gfCNCPoint1[16841] = {X 353.0465, Y 35.4906, Z -1.3333, A 0.000, B 0.000, C 0.000 }
gfCNCPoint1[16842] = {X 354.2270, Y 34.3409, Z -1.3333, A 0.000, B 0.000, C 0.000 }
gfCNCPoint1[16843] = {X 355.2487, Y 33.0481, Z -1.3333, A 0.000, B 0.000, C 0.000 }
gfCNCPoint1[16844] = {X 356.0944, Y 31.6339, Z -1.3333, A 0.000, B 0.000, C 0.000 }
gfCNCPoint1[16845] = {X 356.7500, Y 30.1221, Z -1.3333, A 0.000, B 0.000, C 0.000 }
gfCNCPoint1[16846] = {X 357.2044, Y 28.5381, Z -1.3333, A 0.000, B 0.000, C 0.000 }
gfCNCPoint1[16847] = {X 357.4826, Y 26.8196, Z -1.3333, A 0.000, B 0.000, C 0.000 }
gfCNCPoint1[16848] = {X 357.5960, Y 25.0823, Z -1.3333, A 0.000, B 0.000, C 0.000 }
gfCNCPoint1[16849] = {X 357.5434, Y 23.3422, Z -1.3333, A 0.000, B 0.000, C 0.000 }
gfCNCPoint1[16850] = {X 357.3254, Y 21.6150, Z -1.3333, A 0.000, B 0.000, C 0.000 }
gfCNCPoint1[16851] = {X 356.9800, Y 20.1274, Z -1.3333, A 0.000, B 0.000, C 0.000 }
gfCNCPoint1[16852] = {X 356.4533, Y 18.6940, Z -1.3333, A 0.000, B 0.000, C 0.000 }
gfCNCPoint1[16853] = {X 355.7534, Y 17.3367, Z -1.3333, A 0.000, B 0.000, C 0.000 }
gfCNCPoint1[16854] = {X 354.8909, Y 16.0764, Z -1.3333, A 0.000, B 0.000, C 0.000 }
gfCNCPoint1[16855] = {X 353.9742, Y 15.0542, Z -1.3333, A 0.000, B 0.000, C 0.000 }
gfCNCPoint1[16856] = {X 352.9205, Y 14.1738, Z -1.3333, A 0.000, B 0.000, C 0.000 }
gfCNCPoint1[16857] = {X 351.7516, Y 13.4534, Z -1.3333, A 0.000, B 0.000, C 0.000 }
gfCNCPoint1[16858] = {X 350.4916, Y 12.9079, Z -1.3333, A 0.000, B 0.000, C 0.000 }
gfCNCPoint1[16859] = {X 349.1664, Y 12.5485, Z -1.3333, A 0.000, B 0.000, C 0.000 }
gfCNCPoint1[16860] = {X 347.3712, Y 12.3248, Z -1.3333, A 0.000, B 0.000, C 0.000 }
gfCNCPoint1[16861] = {X 345.5623, Y 12.3395, Z -1.3333, A 0.000, B 0.000, C 0.000 }
gfCNCPoint1[16862] = {X 343.7710, Y 12.5924, Z -1.3333, A 0.000, B 0.000, C 0.000 }
gfCNCPoint1[16863] = {X 342.0287, Y 13.0789, Z -1.3333, A 0.000, B 0.000, C 0.000 }
gfCNCPoint1[16864] = {X 340.3656, Y 13.7908, Z -1.3333, A 0.000, B 0.000, C 0.000 }
gfCNCPoint1[16865] = {X 338.8108, Y 14.7154, Z -1.3333, A 0.000, B 0.000, C 0.000 }
gfCNCPoint1[16866] = {X 338.7172, Y 14.7804, Z -1.3333, A 0.000, B 0.000, C 0.000 }
gfCNCPoint1[16867] = {X 338.6242, Y 14.8461, Z -1.3333, A 0.000, B 0.000, C 0.000 }
gfCNCPoint1[16868] = {X 338.6379, Y 15.0619, Z -1.3333, A 0.000, B 0.000, C 0.000 }
gfCNCPoint1[16869] = {X 338.5598, Y 16.0346, Z -1.3333, A 0.000, B 0.000, C 0.000 }
gfCNCPoint1[16870] = {X 338.2486, Y 16.9596, Z -1.3333, A 0.000, B 0.000, C 0.000 }
gfCNCPoint1[16871] = {X 337.7226, Y 17.7816, Z -1.3333, A 0.000, B 0.000, C 0.000 }
gfCNCPoint1[16872] = {X 337.0132, Y 18.4518, Z -1.3333, A 0.000, B 0.000, C 0.000 }
gfCNCPoint1[16873] = {X 336.3278, Y 18.9560, Z -1.3333, A 0.000, B 0.000, C 0.000 }
gfCNCPoint1[16874] = {X 335.5713, Y 19.3817, Z -1.3333, A 0.000, B 0.000, C 0.000 }
gfCNCPoint1[16875] = {X 334.7407, Y 19.6341, Z -1.3333, A 0.000, B 0.000, C 0.000 }
gfCNCPoint1[16876] = {X 333.8753, Y 19.7014, Z -1.3333, A 0.000, B 0.000, C 0.000 }
gfCNCPoint1[16877] = {X 333.0157, Y 19.5804, Z -1.3333, A 0.000, B 0.000, C 0.000 }
gfCNCPoint1[16878] = {X 332.2025, Y 19.2768, Z -1.3333, A 0.000, B 0.000, C 0.000 }
gfCNCPoint1[16879] = {X 331.4739, Y 18.8049, Z -1.3333, A 0.000, B 0.000, C 0.000 }
gfCNCPoint1[16880] = {X 330.8643, Y 18.1870, Z -1.3333, A 0.000, B 0.000, C 0.000 }
gfCNCPoint1[16881] = {X 330.4023, Y 17.4521, Z -1.3333, A 0.000, B 0.000, C 0.000 }
gfCNCPoint1[16882] = {X 326.8820, Y 10.2103, Z -1.3333, A 0.000, B 0.000, C 0.000 }
gfCNCPoint1[16883] = {X 326.5719, Y 9.3163, Z -1.3333, A 0.000, B 0.000, C 0.000 }
gfCNCPoint1[16884] = {X 326.4804, Y 8.3746, Z -1.3333, A 0.000, B 0.000, C 0.000 }
gfCNCPoint1[16885] = {X 326.6127, Y 7.4376, Z -1.3333, A 0.000, B 0.000, C 0.000 }
gfCNCPoint1[16886] = {X 326.9614, Y 6.5580, Z -1.3333, A 0.000, B 0.000, C 0.000 }
gfCNCPoint1[16887] = {X 327.5070, Y 5.7849, Z -1.3333, A 0.000, B 0.000, C 0.000 }
gfCNCPoint1[16888] = {X 328.2189, Y 5.1616, Z -1.3333, A 0.000, B 0.000, C 0.000 }
gfCNCPoint1[16889] = {X 328.8880, Y 4.7034, Z -1.3333, A 0.000, B 0.000, C 0.000 }
gfCNCPoint1[16890] = {X 329.7043, Y 4.2813, Z -1.3333, A 0.000, B 0.000, C 0.000 }
gfCNCPoint1[16891] = {X 330.5954, Y 4.0567, Z -1.3333, A 0.000, B 0.000, C 0.000 }
gfCNCPoint1[16892] = {X 331.5142, Y 4.0413, Z -1.3333, A 0.000, B 0.000, C 0.000 }
gfCNCPoint1[16893] = {X 332.4122, Y 4.2361, Z -1.3333, A 0.000, B 0.000, C 0.000 }
gfCNCPoint1[16894] = {X 332.5467, Y 4.2834, Z -1.3333, A 0.000, B 0.000, C 0.000 }
gfCNCPoint1[16895] = {X 332.6264, Y 4.2354, Z -1.3333, A 0.000, B 0.000, C 0.000 }
gfCNCPoint1[16896] = {X 332.7062, Y 4.1876, Z -1.3333, A 0.000, B 0.000, C 0.000 }
gfCNCPoint1[16897] = {X 334.1618, Y 3.3772, Z -1.3333, A 0.000, B 0.000, C 0.000 }
gfCNCPoint1[16898] = {X 335.6629, Y 2.6547, Z -1.3333, A 0.000, B 0.000, C 0.000 }
gfCNCPoint1[16899] = {X 336.0092, Y 2.5006, Z -1.3333, A 0.000, B 0.000, C 0.000 }
gfCNCPoint1[16900] = {X 338.0805, Y 1.6925, Z -1.3333, A 0.000, B 0.000, C 0.000 }
gfCNCPoint1[16901] = {X 340.2133, Y 1.0646, Z -1.3333, A 0.000, B 0.000, C 0.000 }
gfCNCPoint1[16902] = {X 342.3920, Y 0.6215, Z -1.3333, A 0.000, B 0.000, C 0.000 }
gfCNCPoint1[16903] = {X 344.6007, Y 0.3665, Z -1.3333, A 0.000, B 0.000, C 0.000 }
gfCNCPoint1[16904] = {X 346.8231, Y 0.3014, Z -1.3333, A 0.000, B 0.000, C 0.000 }
gfCNCPoint1[16905] = {X 349.0429, Y 0.4266, Z -1.3333, A 0.000, B 0.000, C 0.000 }
gfCNCPoint1[16906] = {X 351.2438, Y 0.7414, Z -1.3333, A 0.000, B 0.000, C 0.000 }
gfCNCPoint1[16907] = {X 351.5273, Y 0.7937, Z -1.3333, A 0.000, B 0.000, C 0.000 }
gfCNCPoint1[16908] = {X 352.2677, Y -3.2186, Z -1.3333, A 0.000, B 0.000, C 0.000 }
gfCNCPoint1[16909] = {X 352.2677, Y -3.2186, Z 1.6667, A 0.000, B 0.000, C 0.000 }
gfCNCPoint1[16910] = {X 352.2677, Y -3.2186, Z 11.0000, A 0.000, B 0.000, C 0.000 }
gfCNCPoint1[16911] = {X 606.0428, Y 42.9012, Z 11.0000, A 0.000, B 0.000, C 0.000 }
gfCNCPoint1[16912] = {X 606.0428, Y 42.9012, Z 1.6667, A 0.000, B 0.000, C 0.000 }
gfCNCPoint1[16913] = {X 606.0428, Y 42.9012, Z -1.3333, A 0.000, B 0.000, C 0.000 }
gfCNCPoint1[16914] = {X 603.6965, Y 47.0770, Z -1.3333, A 0.000, B 0.000, C 0.000 }
gfCNCPoint1[16915] = {X 603.6310, Y 47.1895, Z -1.3333, A 0.000, B 0.000, C 0.000 }
gfCNCPoint1[16916] = {X 603.5620, Y 47.2999, Z -1.3333, A 0.000, B 0.000, C 0.000 }
gfCNCPoint1[16917] = {X 603.0356, Y 47.9602, Z -1.3333, A 0.000, B 0.000, C 0.000 }
gfCNCPoint1[16918] = {X 602.3888, Y 48.5030, Z -1.3333, A 0.000, B 0.000, C 0.000 }
gfCNCPoint1[16919] = {X 601.6472, Y 48.9070, Z -1.3333, A 0.000, B 0.000, C 0.000 }
gfCNCPoint1[16920] = {X 600.8403, Y 49.1559, Z -1.3333, A 0.000, B 0.000, C 0.000 }
gfCNCPoint1[16921] = {X 600.0000, Y 49.2400, Z -1.3333, A 0.000, B 0.000, C 0.000 }
gfCNCPoint1[16922] = {X 593.5565, Y 49.2400, Z -1.3333, A 0.000, B 0.000, C 0.000 }
gfCNCPoint1[16923] = {X 592.6130, Y 49.1337, Z -1.3333, A 0.000, B 0.000, C 0.000 }
gfCNCPoint1[16924] = {X 591.7169, Y 48.8201, Z -1.3333, A 0.000, B 0.000, C 0.000 }
gfCNCPoint1[16925] = {X 590.9129, Y 48.3150, Z -1.3333, A 0.000, B 0.000, C 0.000 }
gfCNCPoint1[16926] = {X 590.2416, Y 47.6436, Z -1.3333, A 0.000, B 0.000, C 0.000 }
gfCNCPoint1[16927] = {X 589.7364, Y 46.8397, Z -1.3333, A 0.000, B 0.000, C 0.000 }
gfCNCPoint1[16928] = {X 589.4228, Y 45.9435, Z -1.3333, A 0.000, B 0.000, C 0.000 }
gfCNCPoint1[16929] = {X 589.3165, Y 45.0000, Z -1.3333, A 0.000, B 0.000, C 0.000 }
gfCNCPoint1[16930] = {X 589.3165, Y 44.0647, Z -1.3333, A 0.000, B 0.000, C 0.000 }
gfCNCPoint1[16931] = {X 589.4217, Y 43.1448, Z -1.3333, A 0.000, B 0.000, C 0.000 }
gfCNCPoint1[16932] = {X 589.7219, Y 42.2689, Z -1.3333, A 0.000, B 0.000, C 0.000 }
gfCNCPoint1[16933] = {X 590.2033, Y 41.4779, Z -1.3333, A 0.000, B 0.000, C 0.000 }
gfCNCPoint1[16934] = {X 590.8434, Y 40.8088, Z -1.3333, A 0.000, B 0.000, C 0.000 }
gfCNCPoint1[16935] = {X 590.8437, Y 33.1183, Z -1.3333, A 0.000, B 0.000, C 0.000 }
gfCNCPoint1[16936] = {X 585.3714, Y 46.6218, Z -1.3333, A 0.000, B 0.000, C 0.000 }
gfCNCPoint1[16937] = {X 585.0085, Y 47.3114, Z -1.3333, A 0.000, B 0.000, C 0.000 }
gfCNCPoint1[16938] = {X 584.5255, Y 47.9228, Z -1.3333, A 0.000, B 0.000, C 0.000 }
gfCNCPoint1[16939] = {X 583.9387, Y 48.4356, Z -1.3333, A 0.000, B 0.000, C 0.000 }
gfCNCPoint1[16940] = {X 583.2680, Y 48.8323, Z -1.3333, A 0.000, B 0.000, C 0.000 }
gfCNCPoint1[16941] = {X 582.3418, Y 49.1460, Z -1.3333, A 0.000, B 0.000, C 0.000 }
gfCNCPoint1[16942] = {X 581.3682, Y 49.2391, Z -1.3333, A 0.000, B 0.000, C 0.000 }
gfCNCPoint1[16943] = {X 580.3993, Y 49.1068, Z -1.3333, A 0.000, B 0.000, C 0.000 }
gfCNCPoint1[16944] = {X 579.4864, Y 48.7559, Z -1.3333, A 0.000, B 0.000, C 0.000 }
gfCNCPoint1[16945] = {X 578.6782, Y 48.2052, Z -1.3333, A 0.000, B 0.000, C 0.000 }
gfCNCPoint1[16946] = {X 578.0177, Y 47.4840, Z -1.3333, A 0.000, B 0.000, C 0.000 }
gfCNCPoint1[16947] = {X 577.5400, Y 46.6307, Z -1.3333, A 0.000, B 0.000, C 0.000 }
gfCNCPoint1[16948] = {X 571.9376, Y 32.9313, Z -1.3333, A 0.000, B 0.000, C 0.000 }
gfCNCPoint1[16949] = {X 571.9380, Y 40.8075, Z -1.3333, A 0.000, B 0.000, C 0.000 }
gfCNCPoint1[16950] = {X 572.5762, Y 41.4678, Z -1.3333, A 0.000, B 0.000, C 0.000 }
gfCNCPoint1[16951] = {X 573.0573, Y 42.2500, Z -1.3333, A 0.000, B 0.000, C 0.000 }
gfCNCPoint1[16952] = {X 573.3587, Y 43.1174, Z -1.3333, A 0.000, B 0.000, C 0.000 }
gfCNCPoint1[16953] = {X 573.4663, Y 44.0294, Z -1.3333, A 0.000, B 0.000, C 0.000 }
gfCNCPoint1[16954] = {X 573.4664, Y 45.0000, Z -1.3333, A 0.000, B 0.000, C 0.000 }
gfCNCPoint1[16955] = {X 573.3601, Y 45.9435, Z -1.3333, A 0.000, B 0.000, C 0.000 }
gfCNCPoint1[16956] = {X 573.0465, Y 46.8397, Z -1.3333, A 0.000, B 0.000, C 0.000 }
gfCNCPoint1[16957] = {X 572.5414, Y 47.6436, Z -1.3333, A 0.000, B 0.000, C 0.000 }
gfCNCPoint1[16958] = {X 571.8700, Y 48.3150, Z -1.3333, A 0.000, B 0.000, C 0.000 }
gfCNCPoint1[16959] = {X 571.0661, Y 48.8201, Z -1.3333, A 0.000, B 0.000, C 0.000 }
gfCNCPoint1[16960] = {X 570.1699, Y 49.1337, Z -1.3333, A 0.000, B 0.000, C 0.000 }
gfCNCPoint1[16961] = {X 569.2264, Y 49.2400, Z -1.3333, A 0.000, B 0.000, C 0.000 }
gfCNCPoint1[16962] = {X 562.4443, Y 49.2400, Z -1.3333, A 0.000, B 0.000, C 0.000 }
gfCNCPoint1[16963] = {X 561.5008, Y 49.1337, Z -1.3333, A 0.000, B 0.000, C 0.000 }
gfCNCPoint1[16964] = {X 560.6046, Y 48.8201, Z -1.3333, A 0.000, B 0.000, C 0.000 }
gfCNCPoint1[16965] = {X 559.8007, Y 48.3150, Z -1.3333, A 0.000, B 0.000, C 0.000 }
gfCNCPoint1[16966] = {X 559.1293, Y 47.6436, Z -1.3333, A 0.000, B 0.000, C 0.000 }
gfCNCPoint1[16967] = {X 558.6242, Y 46.8397, Z -1.3333, A 0.000, B 0.000, C 0.000 }
gfCNCPoint1[16968] = {X 558.3106, Y 45.9435, Z -1.3333, A 0.000, B 0.000, C 0.000 }
gfCNCPoint1[16969] = {X 558.2043, Y 45.0000, Z -1.3333, A 0.000, B 0.000, C 0.000 }
gfCNCPoint1[16970] = {X 558.2043, Y 44.0648, Z -1.3333, A 0.000, B 0.000, C 0.000 }
gfCNCPoint1[16971] = {X 558.3092, Y 43.1444, Z -1.3333, A 0.000, B 0.000, C 0.000 }
gfCNCPoint1[16972] = {X 558.6098, Y 42.2682, Z -1.3333, A 0.000, B 0.000, C 0.000 }
gfCNCPoint1[16973] = {X 559.0919, Y 41.4773, Z -1.3333, A 0.000, B 0.000, C 0.000 }
gfCNCPoint1[16974] = {X 559.7330, Y 40.8086, Z -1.3333, A 0.000, B 0.000, C 0.000 }
gfCNCPoint1[16975] = {X 559.7330, Y 9.1939, Z -1.3333, A 0.000, B 0.000, C 0.000 }
gfCNCPoint1[16976] = {X 559.0946, Y 8.5335, Z -1.3333, A 0.000, B 0.000, C 0.000 }
gfCNCPoint1[16977] = {X 558.6134, Y 7.7511, Z -1.3333, A 0.000, B 0.000, C 0.000 }
gfCNCPoint1[16978] = {X 558.3119, Y 6.8834, Z -1.3333, A 0.000, B 0.000, C 0.000 }
gfCNCPoint1[16979] = {X 558.2045, Y 5.9711, Z -1.3333, A 0.000, B 0.000, C 0.000 }
gfCNCPoint1[16980] = {X 558.2043, Y 5.0000, Z -1.3333, A 0.000, B 0.000, C 0.000 }
gfCNCPoint1[16981] = {X 558.3106, Y 4.0565, Z -1.3333, A 0.000, B 0.000, C 0.000 }
gfCNCPoint1[16982] = {X 558.6242, Y 3.1603, Z -1.3333, A 0.000, B 0.000, C 0.000 }
gfCNCPoint1[16983] = {X 559.1293, Y 2.3564, Z -1.3333, A 0.000, B 0.000, C 0.000 }
gfCNCPoint1[16984] = {X 559.8007, Y 1.6850, Z -1.3333, A 0.000, B 0.000, C 0.000 }
gfCNCPoint1[16985] = {X 560.6046, Y 1.1799, Z -1.3333, A 0.000, B 0.000, C 0.000 }
gfCNCPoint1[16986] = {X 561.5008, Y 0.8663, Z -1.3333, A 0.000, B 0.000, C 0.000 }
gfCNCPoint1[16987] = {X 562.4443, Y 0.7600, Z -1.3333, A 0.000, B 0.000, C 0.000 }
gfCNCPoint1[16988] = {X 570.9376, Y 0.7600, Z -1.3333, A 0.000, B 0.000, C 0.000 }
gfCNCPoint1[16989] = {X 571.8810, Y 0.8663, Z -1.3333, A 0.000, B 0.000, C 0.000 }
gfCNCPoint1[16990] = {X 572.7772, Y 1.1799, Z -1.3333, A 0.000, B 0.000, C 0.000 }
gfCNCPoint1[16991] = {X 573.5812, Y 1.6850, Z -1.3333, A 0.000, B 0.000, C 0.000 }
gfCNCPoint1[16992] = {X 574.2525, Y 2.3564, Z -1.3333, A 0.000, B 0.000, C 0.000 }
gfCNCPoint1[16993] = {X 574.7577, Y 3.1603, Z -1.3333, A 0.000, B 0.000, C 0.000 }
gfCNCPoint1[16994] = {X 575.0712, Y 4.0565, Z -1.3333, A 0.000, B 0.000, C 0.000 }
gfCNCPoint1[16995] = {X 575.1776, Y 5.0000, Z -1.3333, A 0.000, B 0.000, C 0.000 }
gfCNCPoint1[16996] = {X 575.1776, Y 5.9342, Z -1.3333, A 0.000, B 0.000, C 0.000 }
gfCNCPoint1[16997] = {X 575.1023, Y 6.7296, Z -1.3333, A 0.000, B 0.000, C 0.000 }
gfCNCPoint1[16998] = {X 574.8791, Y 7.4967, Z -1.3333, A 0.000, B 0.000, C 0.000 }
gfCNCPoint1[16999] = {X 574.5160, Y 8.2083, Z -1.3333, A 0.000, B 0.000, C 0.000 }
gfCNCPoint1[17000] = {X 581.1908, Y 24.5828, Z -1.3333, A 0.000, B 0.000, C 0.000 }
gfCNCPoint1[17001] = {X 587.9351, Y 8.0884, Z -1.3333, A 0.000, B 0.000, C 0.000 }
gfCNCPoint1[17002] = {X 587.6160, Y 7.4203, Z -1.3333, A 0.000, B 0.000, C 0.000 }
gfCNCPoint1[17003] = {X 587.4180, Y 6.7068, Z -1.3333, A 0.000, B 0.000, C 0.000 }
gfCNCPoint1[17004] = {X 587.3471, Y 5.9698, Z -1.3333, A 0.000, B 0.000, C 0.000 }
gfCNCPoint1[17005] = {X 587.3470, Y 5.0000, Z -1.3333, A 0.000, B 0.000, C 0.000 }
gfCNCPoint1[17006] = {X 587.4533, Y 4.0565, Z -1.3333, A 0.000, B 0.000, C 0.000 }
gfCNCPoint1[17007] = {X 587.7668, Y 3.1603, Z -1.3333, A 0.000, B 0.000, C 0.000 }
gfCNCPoint1[17008] = {X 588.2720, Y 2.3564, Z -1.3333, A 0.000, B 0.000, C 0.000 }
gfCNCPoint1[17009] = {X 588.9434, Y 1.6850, Z -1.3333, A 0.000, B 0.000, C 0.000 }
gfCNCPoint1[17010] = {X 589.7473, Y 1.1799, Z -1.3333, A 0.000, B 0.000, C 0.000 }
gfCNCPoint1[17011] = {X 590.6435, Y 0.8663, Z -1.3333, A 0.000, B 0.000, C 0.000 }
gfCNCPoint1[17012] = {X 591.5870, Y 0.7600, Z -1.3333, A 0.000, B 0.000, C 0.000 }
gfCNCPoint1[17013] = {X 600.0000, Y 0.7600, Z -1.3333, A 0.000, B 0.000, C 0.000 }
gfCNCPoint1[17014] = {X 600.8403, Y 0.8441, Z -1.3333, A 0.000, B 0.000, C 0.000 }
gfCNCPoint1[17015] = {X 601.6472, Y 1.0930, Z -1.3333, A 0.000, B 0.000, C 0.000 }
gfCNCPoint1[17016] = {X 602.3888, Y 1.4970, Z -1.3333, A 0.000, B 0.000, C 0.000 }
gfCNCPoint1[17017] = {X 603.0356, Y 2.0398, Z -1.3333, A 0.000, B 0.000, C 0.000 }
gfCNCPoint1[17018] = {X 603.5620, Y 2.7001, Z -1.3333, A 0.000, B 0.000, C 0.000 }
gfCNCPoint1[17019] = {X 603.6310, Y 2.8105, Z -1.3333, A 0.000, B 0.000, C 0.000 }
gfCNCPoint1[17020] = {X 603.6965, Y 2.9230, Z -1.3333, A 0.000, B 0.000, C 0.000 }
gfCNCPoint1[17021] = {X 607.8235, Y 10.2681, Z -1.3333, A 0.000, B 0.000, C 0.000 }
gfCNCPoint1[17022] = {X 607.8235, Y 10.2681, Z 1.6667, A 0.000, B 0.000, C 0.000 }
gfCNCPoint1[17023] = {X 607.8235, Y 10.2681, Z 11.0000, A 0.000, B 0.000, C 0.000 }
gfCNCPoint1[17024] = {X 607.6965, Y 39.1604, Z 11.0000, A 0.000, B 0.000, C 0.000 }
gfCNCPoint1[17025] = {X 607.6965, Y 39.1604, Z 1.6667, A 0.000, B 0.000, C 0.000 }
gfCNCPoint1[17026] = {X 607.6965, Y 39.1604, Z -1.3333, A 0.000, B 0.000, C 0.000 }
gfCNCPoint1[17027] = {X 603.6965, Y 46.9084, Z -1.3333, A 0.000, B 0.000, C 0.000 }
gfCNCPoint1[17028] = {X 603.5999, Y 47.0849, Z -1.3333, A 0.000, B 0.000, C 0.000 }
gfCNCPoint1[17029] = {X 603.4948, Y 47.2565, Z -1.3333, A 0.000, B 0.000, C 0.000 }
gfCNCPoint1[17030] = {X 602.9783, Y 47.9043, Z -1.3333, A 0.000, B 0.000, C 0.000 }
gfCNCPoint1[17031] = {X 602.3437, Y 48.4370, Z -1.3333, A 0.000, B 0.000, C 0.000 }
gfCNCPoint1[17032] = {X 601.6161, Y 48.8332, Z -1.3333, A 0.000, B 0.000, C 0.000 }
gfCNCPoint1[17033] = {X 600.8244, Y 49.0775, Z -1.3333, A 0.000, B 0.000, C 0.000 }
gfCNCPoint1[17034] = {X 600.0000, Y 49.1600, Z -1.3333, A 0.000, B 0.000, C 0.000 }
gfCNCPoint1[17035] = {X 593.5565, Y 49.1600, Z -1.3333, A 0.000, B 0.000, C 0.000 }
gfCNCPoint1[17036] = {X 592.6308, Y 49.0557, Z -1.3333, A 0.000, B 0.000, C 0.000 }
gfCNCPoint1[17037] = {X 591.7516, Y 48.7480, Z -1.3333, A 0.000, B 0.000, C 0.000 }
gfCNCPoint1[17038] = {X 590.9628, Y 48.2524, Z -1.3333, A 0.000, B 0.000, C 0.000 }
gfCNCPoint1[17039] = {X 590.3041, Y 47.5937, Z -1.3333, A 0.000, B 0.000, C 0.000 }
gfCNCPoint1[17040] = {X 589.8085, Y 46.8050, Z -1.3333, A 0.000, B 0.000, C 0.000 }
gfCNCPoint1[17041] = {X 589.5008, Y 45.9257, Z -1.3333, A 0.000, B 0.000, C 0.000 }
gfCNCPoint1[17042] = {X 589.3965, Y 45.0000, Z -1.3333, A 0.000, B 0.000, C 0.000 }
gfCNCPoint1[17043] = {X 589.3965, Y 44.0651, Z -1.3333, A 0.000, B 0.000, C 0.000 }
gfCNCPoint1[17044] = {X 589.5018, Y 43.1533, Z -1.3333, A 0.000, B 0.000, C 0.000 }
gfCNCPoint1[17045] = {X 589.8023, Y 42.2860, Z -1.3333, A 0.000, B 0.000, C 0.000 }
gfCNCPoint1[17046] = {X 590.2838, Y 41.5046, Z -1.3333, A 0.000, B 0.000, C 0.000 }
gfCNCPoint1[17047] = {X 590.9234, Y 40.8463, Z -1.3333, A 0.000, B 0.000, C 0.000 }
gfCNCPoint1[17048] = {X 590.9237, Y 32.7078, Z -1.3333, A 0.000, B 0.000, C 0.000 }
gfCNCPoint1[17049] = {X 585.2975, Y 46.5912, Z -1.3333, A 0.000, B 0.000, C 0.000 }
gfCNCPoint1[17050] = {X 584.9414, Y 47.2678, Z -1.3333, A 0.000, B 0.000, C 0.000 }
gfCNCPoint1[17051] = {X 584.4675, Y 47.8677, Z -1.3333, A 0.000, B 0.000, C 0.000 }
gfCNCPoint1[17052] = {X 583.8918, Y 48.3708, Z -1.3333, A 0.000, B 0.000, C 0.000 }
gfCNCPoint1[17053] = {X 583.2338, Y 48.7600, Z -1.3333, A 0.000, B 0.000, C 0.000 }
gfCNCPoint1[17054] = {X 582.3250, Y 49.0678, Z -1.3333, A 0.000, B 0.000, C 0.000 }
gfCNCPoint1[17055] = {X 581.3699, Y 49.1592, Z -1.3333, A 0.000, B 0.000, C 0.000 }
gfCNCPoint1[17056] = {X 580.4192, Y 49.0293, Z -1.3333, A 0.000, B 0.000, C 0.000 }
gfCNCPoint1[17057] = {X 579.5236, Y 48.6850, Z -1.3333, A 0.000, B 0.000, C 0.000 }
gfCNCPoint1[17058] = {X 578.7306, Y 48.1448, Z -1.3333, A 0.000, B 0.000, C 0.000 }
gfCNCPoint1[17059] = {X 578.0826, Y 47.4372, Z -1.3333, A 0.000, B 0.000, C 0.000 }
gfCNCPoint1[17060] = {X 577.6138, Y 46.5999, Z -1.3333, A 0.000, B 0.000, C 0.000 }
gfCNCPoint1[17061] = {X 571.8576, Y 32.5243, Z -1.3333, A 0.000, B 0.000, C 0.000 }
gfCNCPoint1[17062] = {X 571.8580, Y 40.8459, Z -1.3333, A 0.000, B 0.000, C 0.000 }
gfCNCPoint1[17063] = {X 571.9192, Y 40.8950, Z -1.3333, A 0.000, B 0.000, C 0.000 }
gfCNCPoint1[17064] = {X 572.5325, Y 41.5410, Z -1.3333, A 0.000, B 0.000, C 0.000 }
gfCNCPoint1[17065] = {X 572.9943, Y 42.3027, Z -1.3333, A 0.000, B 0.000, C 0.000 }
gfCNCPoint1[17066] = {X 573.2833, Y 43.1453, Z -1.3333, A 0.000, B 0.000, C 0.000 }
gfCNCPoint1[17067] = {X 573.3863, Y 44.0301, Z -1.3333, A 0.000, B 0.000, C 0.000 }
gfCNCPoint1[17068] = {X 573.3864, Y 45.0000, Z -1.3333, A 0.000, B 0.000, C 0.000 }
gfCNCPoint1[17069] = {X 573.2821, Y 45.9257, Z -1.3333, A 0.000, B 0.000, C 0.000 }
gfCNCPoint1[17070] = {X 572.9745, Y 46.8050, Z -1.3333, A 0.000, B 0.000, C 0.000 }
gfCNCPoint1[17071] = {X 572.4788, Y 47.5937, Z -1.3333, A 0.000, B 0.000, C 0.000 }
gfCNCPoint1[17072] = {X 571.8201, Y 48.2524, Z -1.3333, A 0.000, B 0.000, C 0.000 }
gfCNCPoint1[17073] = {X 571.0314, Y 48.7480, Z -1.3333, A 0.000, B 0.000, C 0.000 }
gfCNCPoint1[17074] = {X 570.1521, Y 49.0557, Z -1.3333, A 0.000, B 0.000, C 0.000 }
gfCNCPoint1[17075] = {X 569.2264, Y 49.1600, Z -1.3333, A 0.000, B 0.000, C 0.000 }
gfCNCPoint1[17076] = {X 562.4443, Y 49.1600, Z -1.3333, A 0.000, B 0.000, C 0.000 }
gfCNCPoint1[17077] = {X 561.5186, Y 49.0557, Z -1.3333, A 0.000, B 0.000, C 0.000 }
gfCNCPoint1[17078] = {X 560.6393, Y 48.7480, Z -1.3333, A 0.000, B 0.000, C 0.000 }
gfCNCPoint1[17079] = {X 559.8506, Y 48.2524, Z -1.3333, A 0.000, B 0.000, C 0.000 }
gfCNCPoint1[17080] = {X 559.1919, Y 47.5937, Z -1.3333, A 0.000, B 0.000, C 0.000 }
gfCNCPoint1[17081] = {X 558.6963, Y 46.8050, Z -1.3333, A 0.000, B 0.000, C 0.000 }
gfCNCPoint1[17082] = {X 558.3886, Y 45.9257, Z -1.3333, A 0.000, B 0.000, C 0.000 }
gfCNCPoint1[17083] = {X 558.2843, Y 45.0000, Z -1.3333, A 0.000, B 0.000, C 0.000 }
gfCNCPoint1[17084] = {X 558.2843, Y 44.0652, Z -1.3333, A 0.000, B 0.000, C 0.000 }
gfCNCPoint1[17085] = {X 558.3893, Y 43.1530, Z -1.3333, A 0.000, B 0.000, C 0.000 }
gfCNCPoint1[17086] = {X 558.6902, Y 42.2854, Z -1.3333, A 0.000, B 0.000, C 0.000 }
gfCNCPoint1[17087] = {X 559.1724, Y 41.5040, Z -1.3333, A 0.000, B 0.000, C 0.000 }
gfCNCPoint1[17088] = {X 559.8130, Y 40.8461, Z -1.3333, A 0.000, B 0.000, C 0.000 }
gfCNCPoint1[17089] = {X 559.8130, Y 9.1561, Z -1.3333, A 0.000, B 0.000, C 0.000 }
gfCNCPoint1[17090] = {X 559.1750, Y 8.5065, Z -1.3333, A 0.000, B 0.000, C 0.000 }
gfCNCPoint1[17091] = {X 558.6937, Y 7.7336, Z -1.3333, A 0.000, B 0.000, C 0.000 }
gfCNCPoint1[17092] = {X 558.3920, Y 6.8746, Z -1.3333, A 0.000, B 0.000, C 0.000 }
gfCNCPoint1[17093] = {X 558.2845, Y 5.9704, Z -1.3333, A 0.000, B 0.000, C 0.000 }
gfCNCPoint1[17094] = {X 558.2843, Y 5.0000, Z -1.3333, A 0.000, B 0.000, C 0.000 }
gfCNCPoint1[17095] = {X 558.3886, Y 4.0743, Z -1.3333, A 0.000, B 0.000, C 0.000 }
gfCNCPoint1[17096] = {X 558.6963, Y 3.1950, Z -1.3333, A 0.000, B 0.000, C 0.000 }
gfCNCPoint1[17097] = {X 559.1919, Y 2.4063, Z -1.3333, A 0.000, B 0.000, C 0.000 }
gfCNCPoint1[17098] = {X 559.8506, Y 1.7476, Z -1.3333, A 0.000, B 0.000, C 0.000 }
gfCNCPoint1[17099] = {X 560.6393, Y 1.2520, Z -1.3333, A 0.000, B 0.000, C 0.000 }
gfCNCPoint1[17100] = {X 561.5186, Y 0.9443, Z -1.3333, A 0.000, B 0.000, C 0.000 }
gfCNCPoint1[17101] = {X 562.4443, Y 0.8400, Z -1.3333, A 0.000, B 0.000, C 0.000 }
gfCNCPoint1[17102] = {X 570.9376, Y 0.8400, Z -1.3333, A 0.000, B 0.000, C 0.000 }
gfCNCPoint1[17103] = {X 571.8632, Y 0.9443, Z -1.3333, A 0.000, B 0.000, C 0.000 }
gfCNCPoint1[17104] = {X 572.7425, Y 1.2520, Z -1.3333, A 0.000, B 0.000, C 0.000 }
gfCNCPoint1[17105] = {X 573.5313, Y 1.7476, Z -1.3333, A 0.000, B 0.000, C 0.000 }
gfCNCPoint1[17106] = {X 574.1900, Y 2.4063, Z -1.3333, A 0.000, B 0.000, C 0.000 }
gfCNCPoint1[17107] = {X 574.6856, Y 3.1950, Z -1.3333, A 0.000, B 0.000, C 0.000 }
gfCNCPoint1[17108] = {X 574.9933, Y 4.0743, Z -1.3333, A 0.000, B 0.000, C 0.000 }
gfCNCPoint1[17109] = {X 575.0976, Y 5.0000, Z -1.3333, A 0.000, B 0.000, C 0.000 }
gfCNCPoint1[17110] = {X 575.0976, Y 5.9342, Z -1.3333, A 0.000, B 0.000, C 0.000 }
gfCNCPoint1[17111] = {X 575.0211, Y 6.7280, Z -1.3333, A 0.000, B 0.000, C 0.000 }
gfCNCPoint1[17112] = {X 574.7945, Y 7.4927, Z -1.3333, A 0.000, B 0.000, C 0.000 }
gfCNCPoint1[17113] = {X 574.4262, Y 8.2001, Z -1.3333, A 0.000, B 0.000, C 0.000 }
gfCNCPoint1[17114] = {X 581.1907, Y 24.7945, Z -1.3333, A 0.000, B 0.000, C 0.000 }
gfCNCPoint1[17115] = {X 588.0242, Y 8.0818, Z -1.3333, A 0.000, B 0.000, C 0.000 }
gfCNCPoint1[17116] = {X 587.7002, Y 7.4169, Z -1.3333, A 0.000, B 0.000, C 0.000 }
gfCNCPoint1[17117] = {X 587.4991, Y 6.7052, Z -1.3333, A 0.000, B 0.000, C 0.000 }
gfCNCPoint1[17118] = {X 587.4271, Y 5.9692, Z -1.3333, A 0.000, B 0.000, C 0.000 }
gfCNCPoint1[17119] = {X 587.4270, Y 5.0000, Z -1.3333, A 0.000, B 0.000, C 0.000 }
gfCNCPoint1[17120] = {X 587.5313, Y 4.0743, Z -1.3333, A 0.000, B 0.000, C 0.000 }
gfCNCPoint1[17121] = {X 587.8389, Y 3.1950, Z -1.3333, A 0.000, B 0.000, C 0.000 }
gfCNCPoint1[17122] = {X 588.3345, Y 2.4063, Z -1.3333, A 0.000, B 0.000, C 0.000 }
gfCNCPoint1[17123] = {X 588.9932, Y 1.7476, Z -1.3333, A 0.000, B 0.000, C 0.000 }
gfCNCPoint1[17124] = {X 589.7820, Y 1.2520, Z -1.3333, A 0.000, B 0.000, C 0.000 }
gfCNCPoint1[17125] = {X 590.6613, Y 0.9443, Z -1.3333, A 0.000, B 0.000, C 0.000 }
gfCNCPoint1[17126] = {X 591.5870, Y 0.8400, Z -1.3333, A 0.000, B 0.000, C 0.000 }
gfCNCPoint1[17127] = {X 600.0000, Y 0.8400, Z -1.3333, A 0.000, B 0.000, C 0.000 }
gfCNCPoint1[17128] = {X 600.8244, Y 0.9225, Z -1.3333, A 0.000, B 0.000, C 0.000 }
gfCNCPoint1[17129] = {X 601.6161, Y 1.1668, Z -1.3333, A 0.000, B 0.000, C 0.000 }
gfCNCPoint1[17130] = {X 602.3437, Y 1.5630, Z -1.3333, A 0.000, B 0.000, C 0.000 }
gfCNCPoint1[17131] = {X 602.9783, Y 2.0957, Z -1.3333, A 0.000, B 0.000, C 0.000 }
gfCNCPoint1[17132] = {X 603.4948, Y 2.7435, Z -1.3333, A 0.000, B 0.000, C 0.000 }
gfCNCPoint1[17133] = {X 603.5999, Y 2.9151, Z -1.3333, A 0.000, B 0.000, C 0.000 }
gfCNCPoint1[17134] = {X 603.6965, Y 3.0916, Z -1.3333, A 0.000, B 0.000, C 0.000 }
gfCNCPoint1[17135] = {X 607.6965, Y 10.8396, Z -1.3333, A 0.000, B 0.000, C 0.000 }
gfCNCPoint1[17136] = {X 607.6965, Y 10.8396, Z 1.6667, A 0.000, B 0.000, C 0.000 }
gfCNCPoint1[17137] = {X 607.6965, Y 10.8396, Z 11.0000, A 0.000, B 0.000, C 0.000 }
gfCNCPoint1[17138] = {X 607.6965, Y 38.1656, Z 11.0000, A 0.000, B 0.000, C 0.000 }
gfCNCPoint1[17139] = {X 607.6965, Y 38.1656, Z 1.6667, A 0.000, B 0.000, C 0.000 }
gfCNCPoint1[17140] = {X 607.6965, Y 38.1656, Z -1.3333, A 0.000, B 0.000, C 0.000 }
gfCNCPoint1[17141] = {X 603.6965, Y 46.7270, Z -1.3333, A 0.000, B 0.000, C 0.000 }
gfCNCPoint1[17142] = {X 603.5703, Y 46.9746, Z -1.3333, A 0.000, B 0.000, C 0.000 }
gfCNCPoint1[17143] = {X 603.4276, Y 47.2131, Z -1.3333, A 0.000, B 0.000, C 0.000 }
gfCNCPoint1[17144] = {X 602.9211, Y 47.8485, Z -1.3333, A 0.000, B 0.000, C 0.000 }
gfCNCPoint1[17145] = {X 602.2986, Y 48.3709, Z -1.3333, A 0.000, B 0.000, C 0.000 }
gfCNCPoint1[17146] = {X 601.5850, Y 48.7595, Z -1.3333, A 0.000, B 0.000, C 0.000 }
gfCNCPoint1[17147] = {X 600.8086, Y 48.9991, Z -1.3333, A 0.000, B 0.000, C 0.000 }
gfCNCPoint1[17148] = {X 600.0000, Y 49.0800, Z -1.3333, A 0.000, B 0.000, C 0.000 }
gfCNCPoint1[17149] = {X 593.5565, Y 49.0800, Z -1.3333, A 0.000, B 0.000, C 0.000 }
gfCNCPoint1[17150] = {X 592.6486, Y 48.9777, Z -1.3333, A 0.000, B 0.000, C 0.000 }
gfCNCPoint1[17151] = {X 591.7863, Y 48.6760, Z -1.3333, A 0.000, B 0.000, C 0.000 }
gfCNCPoint1[17152] = {X 591.0127, Y 48.1899, Z -1.3333, A 0.000, B 0.000, C 0.000 }
gfCNCPoint1[17153] = {X 590.3667, Y 47.5438, Z -1.3333, A 0.000, B 0.000, C 0.000 }
gfCNCPoint1[17154] = {X 589.8806, Y 46.7702, Z -1.3333, A 0.000, B 0.000, C 0.000 }
gfCNCPoint1[17155] = {X 589.5788, Y 45.9079, Z -1.3333, A 0.000, B 0.000, C 0.000 }
gfCNCPoint1[17156] = {X 589.4765, Y 45.0000, Z -1.3333, A 0.000, B 0.000, C 0.000 }
gfCNCPoint1[17157] = {X 589.4765, Y 44.0656, Z -1.3333, A 0.000, B 0.000, C 0.000 }
gfCNCPoint1[17158] = {X 589.5818, Y 43.1620, Z -1.3333, A 0.000, B 0.000, C 0.000 }
gfCNCPoint1[17159] = {X 589.8826, Y 42.3034, Z -1.3333, A 0.000, B 0.000, C 0.000 }
gfCNCPoint1[17160] = {X 590.3643, Y 41.5316, Z -1.3333, A 0.000, B 0.000, C 0.000 }
gfCNCPoint1[17161] = {X 591.0034, Y 40.8842, Z -1.3333, A 0.000, B 0.000, C 0.000 }
gfCNCPoint1[17162] = {X 591.0037, Y 32.2974, Z -1.3333, A 0.000, B 0.000, C 0.000 }
gfCNCPoint1[17163] = {X 585.2236, Y 46.5606, Z -1.3333, A 0.000, B 0.000, C 0.000 }
gfCNCPoint1[17164] = {X 584.8743, Y 47.2242, Z -1.3333, A 0.000, B 0.000, C 0.000 }
gfCNCPoint1[17165] = {X 584.4095, Y 47.8125, Z -1.3333, A 0.000, B 0.000, C 0.000 }
gfCNCPoint1[17166] = {X 583.8449, Y 48.3059, Z -1.3333, A 0.000, B 0.000, C 0.000 }
gfCNCPoint1[17167] = {X 583.1996, Y 48.6877, Z -1.3333, A 0.000, B 0.000, C 0.000 }
gfCNCPoint1[17168] = {X 582.3082, Y 48.9895, Z -1.3333, A 0.000, B 0.000, C 0.000 }
gfCNCPoint1[17169] = {X 581.3715, Y 49.0792, Z -1.3333, A 0.000, B 0.000, C 0.000 }
gfCNCPoint1[17170] = {X 580.4391, Y 48.9518, Z -1.3333, A 0.000, B 0.000, C 0.000 }
gfCNCPoint1[17171] = {X 579.5607, Y 48.6142, Z -1.3333, A 0.000, B 0.000, C 0.000 }
gfCNCPoint1[17172] = {X 578.7830, Y 48.0843, Z -1.3333, A 0.000, B 0.000, C 0.000 }
gfCNCPoint1[17173] = {X 578.1474, Y 47.3903, Z -1.3333, A 0.000, B 0.000, C 0.000 }
gfCNCPoint1[17174] = {X 577.6877, Y 46.5692, Z -1.3333, A 0.000, B 0.000, C 0.000 }
gfCNCPoint1[17175] = {X 571.7775, Y 32.1173, Z -1.3333, A 0.000, B 0.000, C 0.000 }
gfCNCPoint1[17176] = {X 571.7780, Y 40.8843, Z -1.3333, A 0.000, B 0.000, C 0.000 }
gfCNCPoint1[17177] = {X 571.8691, Y 40.9574, Z -1.3333, A 0.000, B 0.000, C 0.000 }
gfCNCPoint1[17178] = {X 572.4700, Y 41.5909, Z -1.3333, A 0.000, B 0.000, C 0.000 }
gfCNCPoint1[17179] = {X 572.9223, Y 42.3376, Z -1.3333, A 0.000, B 0.000, C 0.000 }
gfCNCPoint1[17180] = {X 573.2054, Y 43.1636, Z -1.3333, A 0.000, B 0.000, C 0.000 }
gfCNCPoint1[17181] = {X 573.3063, Y 44.0308, Z -1.3333, A 0.000, B 0.000, C 0.000 }
gfCNCPoint1[17182] = {X 573.3064, Y 45.0000, Z -1.3333, A 0.000, B 0.000, C 0.000 }
gfCNCPoint1[17183] = {X 573.2041, Y 45.9079, Z -1.3333, A 0.000, B 0.000, C 0.000 }
gfCNCPoint1[17184] = {X 572.9024, Y 46.7702, Z -1.3333, A 0.000, B 0.000, C 0.000 }
gfCNCPoint1[17185] = {X 572.4163, Y 47.5438, Z -1.3333, A 0.000, B 0.000, C 0.000 }
gfCNCPoint1[17186] = {X 571.7703, Y 48.1899, Z -1.3333, A 0.000, B 0.000, C 0.000 }
gfCNCPoint1[17187] = {X 570.9967, Y 48.6760, Z -1.3333, A 0.000, B 0.000, C 0.000 }
gfCNCPoint1[17188] = {X 570.1343, Y 48.9777, Z -1.3333, A 0.000, B 0.000, C 0.000 }
gfCNCPoint1[17189] = {X 569.2264, Y 49.0800, Z -1.3333, A 0.000, B 0.000, C 0.000 }
gfCNCPoint1[17190] = {X 562.4443, Y 49.0800, Z -1.3333, A 0.000, B 0.000, C 0.000 }
gfCNCPoint1[17191] = {X 561.5364, Y 48.9777, Z -1.3333, A 0.000, B 0.000, C 0.000 }
gfCNCPoint1[17192] = {X 560.6741, Y 48.6760, Z -1.3333, A 0.000, B 0.000, C 0.000 }
gfCNCPoint1[17193] = {X 559.9005, Y 48.1899, Z -1.3333, A 0.000, B 0.000, C 0.000 }
gfCNCPoint1[17194] = {X 559.2544, Y 47.5438, Z -1.3333, A 0.000, B 0.000, C 0.000 }
gfCNCPoint1[17195] = {X 558.7683, Y 46.7702, Z -1.3333, A 0.000, B 0.000, C 0.000 }
gfCNCPoint1[17196] = {X 558.4666, Y 45.9079, Z -1.3333, A 0.000, B 0.000, C 0.000 }
gfCNCPoint1[17197] = {X 558.3643, Y 45.0000, Z -1.3333, A 0.000, B 0.000, C 0.000 }
gfCNCPoint1[17198] = {X 558.3643, Y 44.0656, Z -1.3333, A 0.000, B 0.000, C 0.000 }
gfCNCPoint1[17199] = {X 558.4615, Y 43.1967, Z -1.3333, A 0.000, B 0.000, C 0.000 }
gfCNCPoint1[17200] = {X 558.7400, Y 42.3679, Z -1.3333, A 0.000, B 0.000, C 0.000 }
gfCNCPoint1[17201] = {X 559.1871, Y 41.6165, Z -1.3333, A 0.000, B 0.000, C 0.000 }
gfCNCPoint1[17202] = {X 559.7828, Y 40.9764, Z -1.3333, A 0.000, B 0.000, C 0.000 }
gfCNCPoint1[17203] = {X 559.8375, Y 40.9298, Z -1.3333, A 0.000, B 0.000, C 0.000 }
gfCNCPoint1[17204] = {X 559.8930, Y 40.8841, Z -1.3333, A 0.000, B 0.000, C 0.000 }
gfCNCPoint1[17205] = {X 559.8930, Y 9.1180, Z -1.3333, A 0.000, B 0.000, C 0.000 }
gfCNCPoint1[17206] = {X 559.8370, Y 9.0723, Z -1.3333, A 0.000, B 0.000, C 0.000 }
gfCNCPoint1[17207] = {X 559.7818, Y 9.0256, Z -1.3333, A 0.000, B 0.000, C 0.000 }
gfCNCPoint1[17208] = {X 559.1890, Y 8.3936, Z -1.3333, A 0.000, B 0.000, C 0.000 }
gfCNCPoint1[17209] = {X 558.7430, Y 7.6508, Z -1.3333, A 0.000, B 0.000, C 0.000 }
gfCNCPoint1[17210] = {X 558.4640, Y 6.8305, Z -1.3333, A 0.000, B 0.000, C 0.000 }
gfCNCPoint1[17211] = {X 558.3645, Y 5.9697, Z -1.3333, A 0.000, B 0.000, C 0.000 }
gfCNCPoint1[17212] = {X 558.3643, Y 5.0000, Z -1.3333, A 0.000, B 0.000, C 0.000 }
gfCNCPoint1[17213] = {X 558.4666, Y 4.0921, Z -1.3333, A 0.000, B 0.000, C 0.000 }
gfCNCPoint1[17214] = {X 558.7683, Y 3.2298, Z -1.3333, A 0.000, B 0.000, C 0.000 }
gfCNCPoint1[17215] = {X 559.2544, Y 2.4562, Z -1.3333, A 0.000, B 0.000, C 0.000 }
gfCNCPoint1[17216] = {X 559.9005, Y 1.8101, Z -1.3333, A 0.000, B 0.000, C 0.000 }
gfCNCPoint1[17217] = {X 560.6741, Y 1.3240, Z -1.3333, A 0.000, B 0.000, C 0.000 }
gfCNCPoint1[17218] = {X 561.5364, Y 1.0223, Z -1.3333, A 0.000, B 0.000, C 0.000 }
gfCNCPoint1[17219] = {X 562.4443, Y 0.9200, Z -1.3333, A 0.000, B 0.000, C 0.000 }
gfCNCPoint1[17220] = {X 570.9376, Y 0.9200, Z -1.3333, A 0.000, B 0.000, C 0.000 }
gfCNCPoint1[17221] = {X 571.8454, Y 1.0223, Z -1.3333, A 0.000, B 0.000, C 0.000 }
gfCNCPoint1[17222] = {X 572.7078, Y 1.3240, Z -1.3333, A 0.000, B 0.000, C 0.000 }
gfCNCPoint1[17223] = {X 573.4814, Y 1.8101, Z -1.3333, A 0.000, B 0.000, C 0.000 }
gfCNCPoint1[17224] = {X 574.1274, Y 2.4562, Z -1.3333, A 0.000, B 0.000, C 0.000 }
gfCNCPoint1[17225] = {X 574.6135, Y 3.2298, Z -1.3333, A 0.000, B 0.000, C 0.000 }
gfCNCPoint1[17226] = {X 574.9153, Y 4.0921, Z -1.3333, A 0.000, B 0.000, C 0.000 }
gfCNCPoint1[17227] = {X 575.0176, Y 5.0000, Z -1.3333, A 0.000, B 0.000, C 0.000 }
gfCNCPoint1[17228] = {X 575.0176, Y 5.9342, Z -1.3333, A 0.000, B 0.000, C 0.000 }
gfCNCPoint1[17229] = {X 574.9499, Y 6.6740, Z -1.3333, A 0.000, B 0.000, C 0.000 }
gfCNCPoint1[17230] = {X 574.7492, Y 7.3893, Z -1.3333, A 0.000, B 0.000, C 0.000 }
gfCNCPoint1[17231] = {X 574.4221, Y 8.0564, Z -1.3333, A 0.000, B 0.000, C 0.000 }
gfCNCPoint1[17232] = {X 574.3778, Y 8.1274, Z -1.3333, A 0.000, B 0.000, C 0.000 }
gfCNCPoint1[17233] = {X 574.3321, Y 8.1975, Z -1.3333, A 0.000, B 0.000, C 0.000 }
gfCNCPoint1[17234] = {X 574.3568, Y 8.2409, Z -1.3333, A 0.000, B 0.000, C 0.000 }
gfCNCPoint1[17235] = {X 581.1906, Y 25.0062, Z -1.3333, A 0.000, B 0.000, C 0.000 }
gfCNCPoint1[17236] = {X 588.1136, Y 8.0746, Z -1.3333, A 0.000, B 0.000, C 0.000 }
gfCNCPoint1[17237] = {X 587.7846, Y 7.4133, Z -1.3333, A 0.000, B 0.000, C 0.000 }
gfCNCPoint1[17238] = {X 587.5802, Y 6.7035, Z -1.3333, A 0.000, B 0.000, C 0.000 }
gfCNCPoint1[17239] = {X 587.5071, Y 5.9685, Z -1.3333, A 0.000, B 0.000, C 0.000 }
gfCNCPoint1[17240] = {X 587.5070, Y 5.0000, Z -1.3333, A 0.000, B 0.000, C 0.000 }
gfCNCPoint1[17241] = {X 587.6092, Y 4.0921, Z -1.3333, A 0.000, B 0.000, C 0.000 }
gfCNCPoint1[17242] = {X 587.9110, Y 3.2298, Z -1.3333, A 0.000, B 0.000, C 0.000 }
gfCNCPoint1[17243] = {X 588.3971, Y 2.4562, Z -1.3333, A 0.000, B 0.000, C 0.000 }
gfCNCPoint1[17244] = {X 589.0431, Y 1.8101, Z -1.3333, A 0.000, B 0.000, C 0.000 }
gfCNCPoint1[17245] = {X 589.8167, Y 1.3240, Z -1.3333, A 0.000, B 0.000, C 0.000 }
gfCNCPoint1[17246] = {X 590.6791, Y 1.0223, Z -1.3333, A 0.000, B 0.000, C 0.000 }
gfCNCPoint1[17247] = {X 591.5870, Y 0.9200, Z -1.3333, A 0.000, B 0.000, C 0.000 }
gfCNCPoint1[17248] = {X 600.0000, Y 0.9200, Z -1.3333, A 0.000, B 0.000, C 0.000 }
gfCNCPoint1[17249] = {X 600.8086, Y 1.0009, Z -1.3333, A 0.000, B 0.000, C 0.000 }
gfCNCPoint1[17250] = {X 601.5850, Y 1.2405, Z -1.3333, A 0.000, B 0.000, C 0.000 }
gfCNCPoint1[17251] = {X 602.2986, Y 1.6291, Z -1.3333, A 0.000, B 0.000, C 0.000 }
gfCNCPoint1[17252] = {X 602.9211, Y 2.1515, Z -1.3333, A 0.000, B 0.000, C 0.000 }
gfCNCPoint1[17253] = {X 603.4276, Y 2.7869, Z -1.3333, A 0.000, B 0.000, C 0.000 }
gfCNCPoint1[17254] = {X 603.5703, Y 3.0254, Z -1.3333, A 0.000, B 0.000, C 0.000 }
gfCNCPoint1[17255] = {X 603.6965, Y 3.2730, Z -1.3333, A 0.000, B 0.000, C 0.000 }
gfCNCPoint1[17256] = {X 607.6965, Y 11.8344, Z -1.3333, A 0.000, B 0.000, C 0.000 }
gfCNCPoint1[17257] = {X 607.6965, Y 11.8344, Z 1.6667, A 0.000, B 0.000, C 0.000 }
gfCNCPoint1[17258] = {X 607.6965, Y 11.8344, Z 11.0000, A 0.000, B 0.000, C 0.000 }
gfCNCPoint1[17259] = {X 607.6965, Y 36.8549, Z 11.0000, A 0.000, B 0.000, C 0.000 }
gfCNCPoint1[17260] = {X 607.6965, Y 36.8549, Z 1.6667, A 0.000, B 0.000, C 0.000 }
gfCNCPoint1[17261] = {X 607.6965, Y 36.8549, Z -1.3333, A 0.000, B 0.000, C 0.000 }
gfCNCPoint1[17262] = {X 603.6965, Y 46.5285, Z -1.3333, A 0.000, B 0.000, C 0.000 }
gfCNCPoint1[17263] = {X 603.5430, Y 46.8567, Z -1.3333, A 0.000, B 0.000, C 0.000 }
gfCNCPoint1[17264] = {X 603.3604, Y 47.1697, Z -1.3333, A 0.000, B 0.000, C 0.000 }
gfCNCPoint1[17265] = {X 602.8638, Y 47.7926, Z -1.3333, A 0.000, B 0.000, C 0.000 }
gfCNCPoint1[17266] = {X 602.2536, Y 48.3048, Z -1.3333, A 0.000, B 0.000, C 0.000 }
gfCNCPoint1[17267] = {X 601.5539, Y 48.6858, Z -1.3333, A 0.000, B 0.000, C 0.000 }
gfCNCPoint1[17268] = {X 600.7927, Y 48.9207, Z -1.3333, A 0.000, B 0.000, C 0.000 }
gfCNCPoint1[17269] = {X 600.0000, Y 49.0000, Z -1.3333, A 0.000, B 0.000, C 0.000 }
gfCNCPoint1[17270] = {X 593.5565, Y 49.0000, Z -1.3333, A 0.000, B 0.000, C 0.000 }
gfCNCPoint1[17271] = {X 592.6664, Y 48.8997, Z -1.3333, A 0.000, B 0.000, C 0.000 }
gfCNCPoint1[17272] = {X 591.8210, Y 48.6039, Z -1.3333, A 0.000, B 0.000, C 0.000 }
gfCNCPoint1[17273] = {X 591.0626, Y 48.1273, Z -1.3333, A 0.000, B 0.000, C 0.000 }
gfCNCPoint1[17274] = {X 590.4292, Y 47.4940, Z -1.3333, A 0.000, B 0.000, C 0.000 }
gfCNCPoint1[17275] = {X 589.9527, Y 46.7355, Z -1.3333, A 0.000, B 0.000, C 0.000 }
gfCNCPoint1[17276] = {X 589.6568, Y 45.8901, Z -1.3333, A 0.000, B 0.000, C 0.000 }
gfCNCPoint1[17277] = {X 589.5565, Y 45.0000, Z -1.3333, A 0.000, B 0.000, C 0.000 }
gfCNCPoint1[17278] = {X 589.5565, Y 44.0660, Z -1.3333, A 0.000, B 0.000, C 0.000 }
gfCNCPoint1[17279] = {X 589.6619, Y 43.1707, Z -1.3333, A 0.000, B 0.000, C 0.000 }
gfCNCPoint1[17280] = {X 589.9630, Y 42.3210, Z -1.3333, A 0.000, B 0.000, C 0.000 }
gfCNCPoint1[17281] = {X 590.4447, Y 41.5590, Z -1.3333, A 0.000, B 0.000, C 0.000 }
gfCNCPoint1[17282] = {X 591.0833, Y 40.9227, Z -1.3333, A 0.000, B 0.000, C 0.000 }
gfCNCPoint1[17283] = {X 591.0854, Y 40.3075, Z -1.3333, A 0.000, B 0.000, C 0.000 }
gfCNCPoint1[17284] = {X 591.0837, Y 32.0423, Z -1.3333, A 0.000, B 0.000, C 0.000 }
gfCNCPoint1[17285] = {X 590.9675, Y 32.1736, Z -1.3333, A 0.000, B 0.000, C 0.000 }
gfCNCPoint1[17286] = {X 590.3133, Y 33.7880, Z -1.3333, A 0.000, B 0.000, C 0.000 }
gfCNCPoint1[17287] = {X 585.1497, Y 46.5300, Z -1.3333, A 0.000, B 0.000, C 0.000 }
gfCNCPoint1[17288] = {X 584.8073, Y 47.1805, Z -1.3333, A 0.000, B 0.000, C 0.000 }
gfCNCPoint1[17289] = {X 584.3516, Y 47.7574, Z -1.3333, A 0.000, B 0.000, C 0.000 }
gfCNCPoint1[17290] = {X 583.7980, Y 48.2411, Z -1.3333, A 0.000, B 0.000, C 0.000 }
gfCNCPoint1[17291] = {X 583.1653, Y 48.6154, Z -1.3333, A 0.000, B 0.000, C 0.000 }
gfCNCPoint1[17292] = {X 582.2878, Y 48.9121, Z -1.3333, A 0.000, B 0.000, C 0.000 }
gfCNCPoint1[17293] = {X 581.3656, Y 48.9990, Z -1.3333, A 0.000, B 0.000, C 0.000 }
gfCNCPoint1[17294] = {X 580.4480, Y 48.8715, Z -1.3333, A 0.000, B 0.000, C 0.000 }
gfCNCPoint1[17295] = {X 579.5845, Y 48.5363, Z -1.3333, A 0.000, B 0.000, C 0.000 }
gfCNCPoint1[17296] = {X 578.8212, Y 48.0115, Z -1.3333, A 0.000, B 0.000, C 0.000 }
gfCNCPoint1[17297] = {X 578.1990, Y 47.3251, Z -1.3333, A 0.000, B 0.000, C 0.000 }
gfCNCPoint1[17298] = {X 577.7515, Y 46.5141, Z -1.3333, A 0.000, B 0.000, C 0.000 }
gfCNCPoint1[17299] = {X 571.6975, Y 31.7102, Z -1.3333, A 0.000, B 0.000, C 0.000 }
gfCNCPoint1[17300] = {X 571.6980, Y 40.9227, Z -1.3333, A 0.000, B 0.000, C 0.000 }
gfCNCPoint1[17301] = {X 571.8369, Y 41.0352, Z -1.3333, A 0.000, B 0.000, C 0.000 }
gfCNCPoint1[17302] = {X 572.4233, Y 41.6618, Z -1.3333, A 0.000, B 0.000, C 0.000 }
gfCNCPoint1[17303] = {X 572.8625, Y 42.3989, Z -1.3333, A 0.000, B 0.000, C 0.000 }
gfCNCPoint1[17304] = {X 573.1344, Y 43.2129, Z -1.3333, A 0.000, B 0.000, C 0.000 }
gfCNCPoint1[17305] = {X 573.2264, Y 44.0660, Z -1.3333, A 0.000, B 0.000, C 0.000 }
gfCNCPoint1[17306] = {X 573.2264, Y 45.0000, Z -1.3333, A 0.000, B 0.000, C 0.000 }
gfCNCPoint1[17307] = {X 573.1261, Y 45.8901, Z -1.3333, A 0.000, B 0.000, C 0.000 }
gfCNCPoint1[17308] = {X 572.8303, Y 46.7355, Z -1.3333, A 0.000, B 0.000, C 0.000 }
gfCNCPoint1[17309] = {X 572.3538, Y 47.4940, Z -1.3333, A 0.000, B 0.000, C 0.000 }
gfCNCPoint1[17310] = {X 571.7204, Y 48.1273, Z -1.3333, A 0.000, B 0.000, C 0.000 }
gfCNCPoint1[17311] = {X 570.9620, Y 48.6039, Z -1.3333, A 0.000, B 0.000, C 0.000 }
gfCNCPoint1[17312] = {X 570.1165, Y 48.8997, Z -1.3333, A 0.000, B 0.000, C 0.000 }
gfCNCPoint1[17313] = {X 569.2264, Y 49.0000, Z -1.3333, A 0.000, B 0.000, C 0.000 }
gfCNCPoint1[17314] = {X 562.4443, Y 49.0000, Z -1.3333, A 0.000, B 0.000, C 0.000 }
gfCNCPoint1[17315] = {X 561.5542, Y 48.8997, Z -1.3333, A 0.000, B 0.000, C 0.000 }
gfCNCPoint1[17316] = {X 560.7088, Y 48.6039, Z -1.3333, A 0.000, B 0.000, C 0.000 }
gfCNCPoint1[17317] = {X 559.9503, Y 48.1273, Z -1.3333, A 0.000, B 0.000, C 0.000 }
gfCNCPoint1[17318] = {X 559.3170, Y 47.4940, Z -1.3333, A 0.000, B 0.000, C 0.000 }
gfCNCPoint1[17319] = {X 558.8404, Y 46.7355, Z -1.3333, A 0.000, B 0.000, C 0.000 }
gfCNCPoint1[17320] = {X 558.5446, Y 45.8901, Z -1.3333, A 0.000, B 0.000, C 0.000 }
gfCNCPoint1[17321] = {X 558.4443, Y 45.0000, Z -1.3333, A 0.000, B 0.000, C 0.000 }
gfCNCPoint1[17322] = {X 558.4443, Y 44.0660, Z -1.3333, A 0.000, B 0.000, C 0.000 }
gfCNCPoint1[17323] = {X 558.5396, Y 43.2140, Z -1.3333, A 0.000, B 0.000, C 0.000 }
gfCNCPoint1[17324] = {X 558.8127, Y 42.4012, Z -1.3333, A 0.000, B 0.000, C 0.000 }
gfCNCPoint1[17325] = {X 559.2511, Y 41.6645, Z -1.3333, A 0.000, B 0.000, C 0.000 }
gfCNCPoint1[17326] = {X 559.8352, Y 41.0368, Z -1.3333, A 0.000, B 0.000, C 0.000 }
gfCNCPoint1[17327] = {X 559.9035, Y 40.9789, Z -1.3333, A 0.000, B 0.000, C 0.000 }
gfCNCPoint1[17328] = {X 559.9730, Y 40.9225, Z -1.3333, A 0.000, B 0.000, C 0.000 }
gfCNCPoint1[17329] = {X 559.9730, Y 9.0793, Z -1.3333, A 0.000, B 0.000, C 0.000 }
gfCNCPoint1[17330] = {X 559.9029, Y 9.0229, Z -1.3333, A 0.000, B 0.000, C 0.000 }
gfCNCPoint1[17331] = {X 559.8340, Y 8.9650, Z -1.3333, A 0.000, B 0.000, C 0.000 }
gfCNCPoint1[17332] = {X 559.2476, Y 8.3384, Z -1.3333, A 0.000, B 0.000, C 0.000 }
gfCNCPoint1[17333] = {X 558.8083, Y 7.6012, Z -1.3333, A 0.000, B 0.000, C 0.000 }
gfCNCPoint1[17334] = {X 558.5363, Y 6.7872, Z -1.3333, A 0.000, B 0.000, C 0.000 }
gfCNCPoint1[17335] = {X 558.4443, Y 5.9339, Z -1.3333, A 0.000, B 0.000, C 0.000 }
gfCNCPoint1[17336] = {X 558.4443, Y 5.0000, Z -1.3333, A 0.000, B 0.000, C 0.000 }
gfCNCPoint1[17337] = {X 558.5446, Y 4.1099, Z -1.3333, A 0.000, B 0.000, C 0.000 }
gfCNCPoint1[17338] = {X 558.8404, Y 3.2645, Z -1.3333, A 0.000, B 0.000, C 0.000 }
gfCNCPoint1[17339] = {X 559.3170, Y 2.5060, Z -1.3333, A 0.000, B 0.000, C 0.000 }
gfCNCPoint1[17340] = {X 559.9503, Y 1.8727, Z -1.3333, A 0.000, B 0.000, C 0.000 }
gfCNCPoint1[17341] = {X 560.7088, Y 1.3961, Z -1.3333, A 0.000, B 0.000, C 0.000 }
gfCNCPoint1[17342] = {X 561.5542, Y 1.1003, Z -1.3333, A 0.000, B 0.000, C 0.000 }
gfCNCPoint1[17343] = {X 562.4443, Y 1.0000, Z -1.3333, A 0.000, B 0.000, C 0.000 }
gfCNCPoint1[17344] = {X 570.9376, Y 1.0000, Z -1.3333, A 0.000, B 0.000, C 0.000 }
gfCNCPoint1[17345] = {X 571.8276, Y 1.1003, Z -1.3333, A 0.000, B 0.000, C 0.000 }
gfCNCPoint1[17346] = {X 572.6731, Y 1.3961, Z -1.3333, A 0.000, B 0.000, C 0.000 }
gfCNCPoint1[17347] = {X 573.4315, Y 1.8727, Z -1.3333, A 0.000, B 0.000, C 0.000 }
gfCNCPoint1[17348] = {X 574.0649, Y 2.5060, Z -1.3333, A 0.000, B 0.000, C 0.000 }
gfCNCPoint1[17349] = {X 574.5414, Y 3.2645, Z -1.3333, A 0.000, B 0.000, C 0.000 }
gfCNCPoint1[17350] = {X 574.8373, Y 4.1099, Z -1.3333, A 0.000, B 0.000, C 0.000 }
gfCNCPoint1[17351] = {X 574.9376, Y 5.0000, Z -1.3333, A 0.000, B 0.000, C 0.000 }
gfCNCPoint1[17352] = {X 574.9372, Y 5.9858, Z -1.3333, A 0.000, B 0.000, C 0.000 }
gfCNCPoint1[17353] = {X 574.8648, Y 6.6933, Z -1.3333, A 0.000, B 0.000, C 0.000 }
gfCNCPoint1[17354] = {X 574.6683, Y 7.3769, Z -1.3333, A 0.000, B 0.000, C 0.000 }
gfCNCPoint1[17355] = {X 574.3538, Y 8.0148, Z -1.3333, A 0.000, B 0.000, C 0.000 }
gfCNCPoint1[17356] = {X 574.2915, Y 8.1137, Z -1.3333, A 0.000, B 0.000, C 0.000 }
gfCNCPoint1[17357] = {X 574.2264, Y 8.2108, Z -1.3333, A 0.000, B 0.000, C 0.000 }
gfCNCPoint1[17358] = {X 574.2601, Y 8.2360, Z -1.3333, A 0.000, B 0.000, C 0.000 }
gfCNCPoint1[17359] = {X 574.2828, Y 8.2713, Z -1.3333, A 0.000, B 0.000, C 0.000 }
gfCNCPoint1[17360] = {X 574.9161, Y 9.8091, Z -1.3333, A 0.000, B 0.000, C 0.000 }
gfCNCPoint1[17361] = {X 581.1904, Y 25.2179, Z -1.3333, A 0.000, B 0.000, C 0.000 }
gfCNCPoint1[17362] = {X 588.2031, Y 8.0670, Z -1.3333, A 0.000, B 0.000, C 0.000 }
gfCNCPoint1[17363] = {X 587.8648, Y 7.3989, Z -1.3333, A 0.000, B 0.000, C 0.000 }
gfCNCPoint1[17364] = {X 587.6570, Y 6.6795, Z -1.3333, A 0.000, B 0.000, C 0.000 }
gfCNCPoint1[17365] = {X 587.5870, Y 5.9339, Z -1.3333, A 0.000, B 0.000, C 0.000 }
gfCNCPoint1[17366] = {X 587.5870, Y 5.0000, Z -1.3333, A 0.000, B 0.000, C 0.000 }
gfCNCPoint1[17367] = {X 587.6872, Y 4.1099, Z -1.3333, A 0.000, B 0.000, C 0.000 }
gfCNCPoint1[17368] = {X 587.9831, Y 3.2645, Z -1.3333, A 0.000, B 0.000, C 0.000 }
gfCNCPoint1[17369] = {X 588.4596, Y 2.5060, Z -1.3333, A 0.000, B 0.000, C 0.000 }
gfCNCPoint1[17370] = {X 589.0930, Y 1.8727, Z -1.3333, A 0.000, B 0.000, C 0.000 }
gfCNCPoint1[17371] = {X 589.8514, Y 1.3961, Z -1.3333, A 0.000, B 0.000, C 0.000 }
gfCNCPoint1[17372] = {X 590.6969, Y 1.1003, Z -1.3333, A 0.000, B 0.000, C 0.000 }
gfCNCPoint1[17373] = {X 591.5870, Y 1.0000, Z -1.3333, A 0.000, B 0.000, C 0.000 }
gfCNCPoint1[17374] = {X 600.0000, Y 1.0000, Z -1.3333, A 0.000, B 0.000, C 0.000 }
gfCNCPoint1[17375] = {X 600.7927, Y 1.0793, Z -1.3333, A 0.000, B 0.000, C 0.000 }
gfCNCPoint1[17376] = {X 601.5539, Y 1.3142, Z -1.3333, A 0.000, B 0.000, C 0.000 }
gfCNCPoint1[17377] = {X 602.2536, Y 1.6952, Z -1.3333, A 0.000, B 0.000, C 0.000 }
gfCNCPoint1[17378] = {X 602.8638, Y 2.2074, Z -1.3333, A 0.000, B 0.000, C 0.000 }
gfCNCPoint1[17379] = {X 603.3604, Y 2.8303, Z -1.3333, A 0.000, B 0.000, C 0.000 }
gfCNCPoint1[17380] = {X 603.5430, Y 3.1433, Z -1.3333, A 0.000, B 0.000, C 0.000 }
gfCNCPoint1[17381] = {X 603.6965, Y 3.4715, Z -1.3333, A 0.000, B 0.000, C 0.000 }
gfCNCPoint1[17382] = {X 607.6965, Y 13.1451, Z -1.3333, A 0.000, B 0.000, C 0.000 }
gfCNCPoint1[17383] = {X 607.6965, Y 13.1451, Z 1.6667, A 0.000, B 0.000, C 0.000 }
gfCNCPoint1[17384] = {X 607.6965, Y 13.1451, Z 11.0000, A 0.000, B 0.000, C 0.000 }
gfCNCPoint1[17385] = {X 256.2409, Y 19.7797, Z 11.0000, A 0.000, B 0.000, C 0.000 }
gfCNCPoint1[17386] = {X 256.2409, Y 19.7797, Z 2.5000, A 0.000, B 0.000, C 0.000 }
gfCNCPoint1[17387] = {X 251.5292, Y 19.7797, Z 1.2375, A 0.000, B 0.000, C 0.000 }
gfCNCPoint1[17388] = {X 250.8347, Y 19.7906, Z 1.0514, A 0.000, B 0.000, C 0.000 }
gfCNCPoint1[17389] = {X 250.1801, Y 19.7923, Z 0.8760, A 0.000, B 0.000, C 0.000 }
gfCNCPoint1[17390] = {X 249.4963, Y 19.8904, Z 0.6909, A 0.000, B 0.000, C 0.000 }
gfCNCPoint1[17391] = {X 248.8451, Y 20.0787, Z 0.5093, A 0.000, B 0.000, C 0.000 }
gfCNCPoint1[17392] = {X 248.7079, Y 20.1100, Z 0.4715, A 0.000, B 0.000, C 0.000 }
gfCNCPoint1[17393] = {X 248.6531, Y 20.1613, Z 0.4514, A 0.000, B 0.000, C 0.000 }
gfCNCPoint1[17394] = {X 248.6131, Y 20.2962, Z 0.4137, A 0.000, B 0.000, C 0.000 }
gfCNCPoint1[17395] = {X 248.4740, Y 20.7643, Z 0.2829, A 0.000, B 0.000, C 0.000 }
gfCNCPoint1[17396] = {X 248.4440, Y 21.8685, Z -0.0131, A 0.000, B 0.000, C 0.000 }
gfCNCPoint1[17397] = {X 248.5574, Y 22.3435, Z -0.1439, A 0.000, B 0.000, C 0.000 }
gfCNCPoint1[17398] = {X 248.8704, Y 22.4376, Z -0.2315, A 0.000, B 0.000, C 0.000 }
gfCNCPoint1[17399] = {X 249.1960, Y 22.4650, Z -0.3191, A 0.000, B 0.000, C 0.000 }
gfCNCPoint1[17400] = {X 250.4374, Y 22.5694, Z -0.6529, A 0.000, B 0.000, C 0.000 }
gfCNCPoint1[17401] = {X 251.6873, Y 22.5560, Z -0.9878, A 0.000, B 0.000, C 0.000 }
gfCNCPoint1[17402] = {X 252.9769, Y 22.5560, Z -1.3333, A 0.000, B 0.000, C 0.000 }
gfCNCPoint1[17403] = {X 257.4115, Y 22.5560, Z -1.3333, A 0.000, B 0.000, C 0.000 }
gfCNCPoint1[17404] = {X 257.4115, Y 19.7797, Z -1.3333, A 0.000, B 0.000, C 0.000 }
gfCNCPoint1[17405] = {X 251.5292, Y 19.7797, Z -1.3333, A 0.000, B 0.000, C 0.000 }
gfCNCPoint1[17406] = {X 250.8347, Y 19.7906, Z -1.3333, A 0.000, B 0.000, C 0.000 }
gfCNCPoint1[17407] = {X 249.8297, Y 19.8641, Z -1.3333, A 0.000, B 0.000, C 0.000 }
gfCNCPoint1[17408] = {X 248.8451, Y 20.0787, Z -1.3333, A 0.000, B 0.000, C 0.000 }
gfCNCPoint1[17409] = {X 248.6996, Y 20.1560, Z -1.3333, A 0.000, B 0.000, C 0.000 }
gfCNCPoint1[17410] = {X 248.6131, Y 20.2962, Z -1.3333, A 0.000, B 0.000, C 0.000 }
gfCNCPoint1[17411] = {X 248.4750, Y 20.9719, Z -1.3333, A 0.000, B 0.000, C 0.000 }
gfCNCPoint1[17412] = {X 248.4562, Y 21.6613, Z -1.3333, A 0.000, B 0.000, C 0.000 }
gfCNCPoint1[17413] = {X 248.5574, Y 22.3435, Z -1.3333, A 0.000, B 0.000, C 0.000 }
gfCNCPoint1[17414] = {X 248.8736, Y 22.4208, Z -1.3333, A 0.000, B 0.000, C 0.000 }
gfCNCPoint1[17415] = {X 249.1960, Y 22.4650, Z -1.3333, A 0.000, B 0.000, C 0.000 }
gfCNCPoint1[17416] = {X 250.4406, Y 22.5400, Z -1.3333, A 0.000, B 0.000, C 0.000 }
gfCNCPoint1[17417] = {X 251.6873, Y 22.5560, Z -1.3333, A 0.000, B 0.000, C 0.000 }
gfCNCPoint1[17418] = {X 252.9769, Y 22.5560, Z -1.3333, A 0.000, B 0.000, C 0.000 }
gfCNCPoint1[17419] = {X 248.9921, Y 22.2874, Z -1.3333, A 0.000, B 0.000, C 0.000 }
gfCNCPoint1[17420] = {X 252.9769, Y 22.6360, Z -1.3333, A 0.000, B 0.000, C 0.000 }
gfCNCPoint1[17421] = {X 257.4915, Y 22.6360, Z -1.3333, A 0.000, B 0.000, C 0.000 }
gfCNCPoint1[17422] = {X 257.4915, Y 19.6997, Z -1.3333, A 0.000, B 0.000, C 0.000 }
gfCNCPoint1[17423] = {X 251.5286, Y 19.6997, Z -1.3333, A 0.000, B 0.000, C 0.000 }
gfCNCPoint1[17424] = {X 250.8365, Y 19.7106, Z -1.3333, A 0.000, B 0.000, C 0.000 }
gfCNCPoint1[17425] = {X 249.8259, Y 19.7842, Z -1.3333, A 0.000, B 0.000, C 0.000 }
gfCNCPoint1[17426] = {X 248.8355, Y 19.9989, Z -1.3333, A 0.000, B 0.000, C 0.000 }
gfCNCPoint1[17427] = {X 248.6480, Y 20.0948, Z -1.3333, A 0.000, B 0.000, C 0.000 }
gfCNCPoint1[17428] = {X 248.5364, Y 20.2734, Z -1.3333, A 0.000, B 0.000, C 0.000 }
gfCNCPoint1[17429] = {X 248.3938, Y 20.9779, Z -1.3333, A 0.000, B 0.000, C 0.000 }
gfCNCPoint1[17430] = {X 248.3783, Y 21.6966, Z -1.3333, A 0.000, B 0.000, C 0.000 }
gfCNCPoint1[17431] = {X 248.4905, Y 22.4065, Z -1.3333, A 0.000, B 0.000, C 0.000 }
gfCNCPoint1[17432] = {X 248.8361, Y 22.4951, Z -1.3333, A 0.000, B 0.000, C 0.000 }
gfCNCPoint1[17433] = {X 249.1893, Y 22.5447, Z -1.3333, A 0.000, B 0.000, C 0.000 }
gfCNCPoint1[17434] = {X 250.4364, Y 22.6199, Z -1.3333, A 0.000, B 0.000, C 0.000 }
gfCNCPoint1[17435] = {X 251.6856, Y 22.6360, Z -1.3333, A 0.000, B 0.000, C 0.000 }
gfCNCPoint1[17436] = {X 252.9769, Y 22.6360, Z -1.3333, A 0.000, B 0.000, C 0.000 }
gfCNCPoint1[17437] = {X 256.9616, Y 22.2874, Z -1.3333, A 0.000, B 0.000, C 0.000 }
gfCNCPoint1[17438] = {X 248.9921, Y 22.3674, Z -1.3333, A 0.000, B 0.000, C 0.000 }
gfCNCPoint1[17439] = {X 252.9769, Y 22.7160, Z -1.3333, A 0.000, B 0.000, C 0.000 }
gfCNCPoint1[17440] = {X 257.5715, Y 22.7160, Z -1.3333, A 0.000, B 0.000, C 0.000 }
gfCNCPoint1[17441] = {X 257.5715, Y 19.6197, Z -1.3333, A 0.000, B 0.000, C 0.000 }
gfCNCPoint1[17442] = {X 251.5280, Y 19.6197, Z -1.3333, A 0.000, B 0.000, C 0.000 }
gfCNCPoint1[17443] = {X 250.8358, Y 19.6306, Z -1.3333, A 0.000, B 0.000, C 0.000 }
gfCNCPoint1[17444] = {X 249.8156, Y 19.7049, Z -1.3333, A 0.000, B 0.000, C 0.000 }
gfCNCPoint1[17445] = {X 248.8159, Y 19.9213, Z -1.3333, A 0.000, B 0.000, C 0.000 }
gfCNCPoint1[17446] = {X 248.5926, Y 20.0371, Z -1.3333, A 0.000, B 0.000, C 0.000 }
gfCNCPoint1[17447] = {X 248.4597, Y 20.2506, Z -1.3333, A 0.000, B 0.000, C 0.000 }
gfCNCPoint1[17448] = {X 248.3127, Y 20.9838, Z -1.3333, A 0.000, B 0.000, C 0.000 }
gfCNCPoint1[17449] = {X 248.3006, Y 21.7315, Z -1.3333, A 0.000, B 0.000, C 0.000 }
gfCNCPoint1[17450] = {X 248.4239, Y 22.4691, Z -1.3333, A 0.000, B 0.000, C 0.000 }
gfCNCPoint1[17451] = {X 248.7987, Y 22.5692, Z -1.3333, A 0.000, B 0.000, C 0.000 }
gfCNCPoint1[17452] = {X 249.1826, Y 22.6244, Z -1.3333, A 0.000, B 0.000, C 0.000 }
gfCNCPoint1[17453] = {X 250.4333, Y 22.6998, Z -1.3333, A 0.000, B 0.000, C 0.000 }
gfCNCPoint1[17454] = {X 251.6860, Y 22.7160, Z -1.3333, A 0.000, B 0.000, C 0.000 }
gfCNCPoint1[17455] = {X 252.9769, Y 22.7160, Z -1.3333, A 0.000, B 0.000, C 0.000 }
gfCNCPoint1[17456] = {X 256.9616, Y 22.3674, Z -1.3333, A 0.000, B 0.000, C 0.000 }
gfCNCPoint1[17457] = {X 248.9921, Y 22.4474, Z -1.3333, A 0.000, B 0.000, C 0.000 }
gfCNCPoint1[17458] = {X 252.9769, Y 22.7960, Z -1.3333, A 0.000, B 0.000, C 0.000 }
gfCNCPoint1[17459] = {X 257.6515, Y 22.7960, Z -1.3333, A 0.000, B 0.000, C 0.000 }
gfCNCPoint1[17460] = {X 257.6515, Y 19.5397, Z -1.3333, A 0.000, B 0.000, C 0.000 }
gfCNCPoint1[17461] = {X 251.5274, Y 19.5397, Z -1.3333, A 0.000, B 0.000, C 0.000 }
gfCNCPoint1[17462] = {X 250.8351, Y 19.5506, Z -1.3333, A 0.000, B 0.000, C 0.000 }
gfCNCPoint1[17463] = {X 249.8053, Y 19.6255, Z -1.3333, A 0.000, B 0.000, C 0.000 }
gfCNCPoint1[17464] = {X 248.7962, Y 19.8437, Z -1.3333, A 0.000, B 0.000, C 0.000 }
gfCNCPoint1[17465] = {X 248.5372, Y 19.9794, Z -1.3333, A 0.000, B 0.000, C 0.000 }
gfCNCPoint1[17466] = {X 248.3830, Y 20.2278, Z -1.3333, A 0.000, B 0.000, C 0.000 }
gfCNCPoint1[17467] = {X 248.2316, Y 20.9896, Z -1.3333, A 0.000, B 0.000, C 0.000 }
gfCNCPoint1[17468] = {X 248.2231, Y 21.7662, Z -1.3333, A 0.000, B 0.000, C 0.000 }
gfCNCPoint1[17469] = {X 248.3577, Y 22.5311, Z -1.3333, A 0.000, B 0.000, C 0.000 }
gfCNCPoint1[17470] = {X 248.7614, Y 22.6431, Z -1.3333, A 0.000, B 0.000, C 0.000 }
gfCNCPoint1[17471] = {X 249.1759, Y 22.7041, Z -1.3333, A 0.000, B 0.000, C 0.000 }
gfCNCPoint1[17472] = {X 250.4301, Y 22.7798, Z -1.3333, A 0.000, B 0.000, C 0.000 }
gfCNCPoint1[17473] = {X 251.6865, Y 22.7960, Z -1.3333, A 0.000, B 0.000, C 0.000 }
gfCNCPoint1[17474] = {X 252.9769, Y 22.7960, Z -1.3333, A 0.000, B 0.000, C 0.000 }
gfCNCPoint1[17475] = {X 256.9616, Y 22.4474, Z -1.3333, A 0.000, B 0.000, C 0.000 }
gfCNCPoint1[17476] = {X 248.9921, Y 22.5274, Z -1.3333, A 0.000, B 0.000, C 0.000 }
gfCNCPoint1[17477] = {X 252.9769, Y 22.8760, Z -1.3333, A 0.000, B 0.000, C 0.000 }
gfCNCPoint1[17478] = {X 257.7315, Y 22.8760, Z -1.3333, A 0.000, B 0.000, C 0.000 }
gfCNCPoint1[17479] = {X 257.7315, Y 19.4597, Z -1.3333, A 0.000, B 0.000, C 0.000 }
gfCNCPoint1[17480] = {X 251.5267, Y 19.4597, Z -1.3333, A 0.000, B 0.000, C 0.000 }
gfCNCPoint1[17481] = {X 250.8344, Y 19.4706, Z -1.3333, A 0.000, B 0.000, C 0.000 }
gfCNCPoint1[17482] = {X 249.7949, Y 19.5462, Z -1.3333, A 0.000, B 0.000, C 0.000 }
gfCNCPoint1[17483] = {X 248.7762, Y 19.7662, Z -1.3333, A 0.000, B 0.000, C 0.000 }
gfCNCPoint1[17484] = {X 248.4816, Y 19.9218, Z -1.3333, A 0.000, B 0.000, C 0.000 }
gfCNCPoint1[17485] = {X 248.3063, Y 20.2051, Z -1.3333, A 0.000, B 0.000, C 0.000 }
gfCNCPoint1[17486] = {X 248.1513, Y 20.9889, Z -1.3333, A 0.000, B 0.000, C 0.000 }
gfCNCPoint1[17487] = {X 248.1446, Y 21.7878, Z -1.3333, A 0.000, B 0.000, C 0.000 }
gfCNCPoint1[17488] = {X 248.2866, Y 22.5741, Z -1.3333, A 0.000, B 0.000, C 0.000 }
gfCNCPoint1[17489] = {X 248.3053, Y 22.5975, Z -1.3333, A 0.000, B 0.000, C 0.000 }
gfCNCPoint1[17490] = {X 248.3316, Y 22.6067, Z -1.3333, A 0.000, B 0.000, C 0.000 }
gfCNCPoint1[17491] = {X 248.7449, Y 22.7214, Z -1.3333, A 0.000, B 0.000, C 0.000 }
gfCNCPoint1[17492] = {X 249.1692, Y 22.7838, Z -1.3333, A 0.000, B 0.000, C 0.000 }
gfCNCPoint1[17493] = {X 250.4270, Y 22.8597, Z -1.3333, A 0.000, B 0.000, C 0.000 }
gfCNCPoint1[17494] = {X 251.6869, Y 22.8760, Z -1.3333, A 0.000, B 0.000, C 0.000 }
gfCNCPoint1[17495] = {X 252.9769, Y 22.8760, Z -1.3333, A 0.000, B 0.000, C 0.000 }
gfCNCPoint1[17496] = {X 256.9616, Y 22.5274, Z -1.3333, A 0.000, B 0.000, C 0.000 }
gfCNCPoint1[17497] = {X 248.9921, Y 22.6074, Z -1.3333, A 0.000, B 0.000, C 0.000 }
gfCNCPoint1[17498] = {X 252.9769, Y 22.9560, Z -1.3333, A 0.000, B 0.000, C 0.000 }
gfCNCPoint1[17499] = {X 257.8115, Y 22.9560, Z -1.3333, A 0.000, B 0.000, C 0.000 }
gfCNCPoint1[17500] = {X 257.8099, Y 19.3797, Z -1.3333, A 0.000, B 0.000, C 0.000 }
gfCNCPoint1[17501] = {X 251.5261, Y 19.3797, Z -1.3333, A 0.000, B 0.000, C 0.000 }
gfCNCPoint1[17502] = {X 250.8336, Y 19.3906, Z -1.3333, A 0.000, B 0.000, C 0.000 }
gfCNCPoint1[17503] = {X 249.7845, Y 19.4669, Z -1.3333, A 0.000, B 0.000, C 0.000 }
gfCNCPoint1[17504] = {X 248.7562, Y 19.6887, Z -1.3333, A 0.000, B 0.000, C 0.000 }
gfCNCPoint1[17505] = {X 248.4261, Y 19.8642, Z -1.3333, A 0.000, B 0.000, C 0.000 }
gfCNCPoint1[17506] = {X 248.2296, Y 20.1823, Z -1.3333, A 0.000, B 0.000, C 0.000 }
gfCNCPoint1[17507] = {X 248.0711, Y 20.9862, Z -1.3333, A 0.000, B 0.000, C 0.000 }
gfCNCPoint1[17508] = {X 248.0659, Y 21.8055, Z -1.3333, A 0.000, B 0.000, C 0.000 }
gfCNCPoint1[17509] = {X 248.2140, Y 22.6114, Z -1.3333, A 0.000, B 0.000, C 0.000 }
gfCNCPoint1[17510] = {X 248.2570, Y 22.6652, Z -1.3333, A 0.000, B 0.000, C 0.000 }
gfCNCPoint1[17511] = {X 248.7032, Y 22.7942, Z -1.3333, A 0.000, B 0.000, C 0.000 }
gfCNCPoint1[17512] = {X 249.1625, Y 22.8636, Z -1.3333, A 0.000, B 0.000, C 0.000 }
gfCNCPoint1[17513] = {X 250.4238, Y 22.9397, Z -1.3333, A 0.000, B 0.000, C 0.000 }
gfCNCPoint1[17514] = {X 251.6873, Y 22.9560, Z -1.3333, A 0.000, B 0.000, C 0.000 }
gfCNCPoint1[17515] = {X 252.9769, Y 22.9560, Z -1.3333, A 0.000, B 0.000, C 0.000 }
gfCNCPoint1[17516] = {X 256.9616, Y 22.6074, Z -1.3333, A 0.000, B 0.000, C 0.000 }
gfCNCPoint1[17517] = {X 256.9616, Y 22.6074, Z 1.6667, A 0.000, B 0.000, C 0.000 }
gfCNCPoint1[17518] = {X 256.9616, Y 22.6074, Z 11.0000, A 0.000, B 0.000, C 0.000 }
gfCNCPoint1[17519] = {X 188.4934, Y 19.4645, Z 11.0000, A 0.000, B 0.000, C 0.000 }
gfCNCPoint1[17520] = {X 188.4934, Y 19.4645, Z 2.5000, A 0.000, B 0.000, C 0.000 }
gfCNCPoint1[17521] = {X 188.3890, Y 19.4275, Z 2.4703, A 0.000, B 0.000, C 0.000 }
gfCNCPoint1[17522] = {X 187.7714, Y 19.3586, Z 2.3038, A 0.000, B 0.000, C 0.000 }
gfCNCPoint1[17523] = {X 186.9109, Y 19.2586, Z 2.0717, A 0.000, B 0.000, C 0.000 }
gfCNCPoint1[17524] = {X 184.5930, Y 19.3661, Z 1.4500, A 0.000, B 0.000, C 0.000 }
gfCNCPoint1[17525] = {X 183.7431, Y 19.5458, Z 1.2172, A 0.000, B 0.000, C 0.000 }
gfCNCPoint1[17526] = {X 183.0408, Y 19.6899, Z 1.0251, A 0.000, B 0.000, C 0.000 }
gfCNCPoint1[17527] = {X 182.0263, Y 20.0592, Z 0.7358, A 0.000, B 0.000, C 0.000 }
gfCNCPoint1[17528] = {X 181.3956, Y 20.4002, Z 0.5437, A 0.000, B 0.000, C 0.000 }
gfCNCPoint1[17529] = {X 181.3398, Y 20.9118, Z 0.4058, A 0.000, B 0.000, C 0.000 }
gfCNCPoint1[17530] = {X 180.8638, Y 22.1280, Z 0.0558, A 0.000, B 0.000, C 0.000 }
gfCNCPoint1[17531] = {X 180.5575, Y 22.5416, Z -0.0821, A 0.000, B 0.000, C 0.000 }
gfCNCPoint1[17532] = {X 182.2902, Y 22.3356, Z -0.5496, A 0.000, B 0.000, C 0.000 }
gfCNCPoint1[17533] = {X 182.5945, Y 22.3109, Z -0.6314, A 0.000, B 0.000, C 0.000 }
gfCNCPoint1[17534] = {X 184.3414, Y 22.2348, Z -1.0999, A 0.000, B 0.000, C 0.000 }
gfCNCPoint1[17535] = {X 184.7767, Y 22.2198, Z -1.2166, A 0.000, B 0.000, C 0.000 }
gfCNCPoint1[17536] = {X 185.2118, Y 22.2014, Z -1.3333, A 0.000, B 0.000, C 0.000 }
gfCNCPoint1[17537] = {X 187.5427, Y 22.0788, Z -1.3333, A 0.000, B 0.000, C 0.000 }
gfCNCPoint1[17538] = {X 189.8705, Y 21.9078, Z -1.3333, A 0.000, B 0.000, C 0.000 }
gfCNCPoint1[17539] = {X 190.4723, Y 21.8322, Z -1.3333, A 0.000, B 0.000, C 0.000 }
gfCNCPoint1[17540] = {X 191.0596, Y 21.6807, Z -1.3333, A 0.000, B 0.000, C 0.000 }
gfCNCPoint1[17541] = {X 191.0694, Y 21.1637, Z -1.3333, A 0.000, B 0.000, C 0.000 }
gfCNCPoint1[17542] = {X 190.8731, Y 20.6854, Z -1.3333, A 0.000, B 0.000, C 0.000 }
gfCNCPoint1[17543] = {X 190.5029, Y 20.3243, Z -1.3333, A 0.000, B 0.000, C 0.000 }
gfCNCPoint1[17544] = {X 189.6453, Y 19.8642, Z -1.3333, A 0.000, B 0.000, C 0.000 }
gfCNCPoint1[17545] = {X 188.7277, Y 19.5397, Z -1.3333, A 0.000, B 0.000, C 0.000 }
gfCNCPoint1[17546] = {X 187.7714, Y 19.3586, Z -1.3333, A 0.000, B 0.000, C 0.000 }
gfCNCPoint1[17547] = {X 186.4245, Y 19.2755, Z -1.3333, A 0.000, B 0.000, C 0.000 }
gfCNCPoint1[17548] = {X 185.0765, Y 19.3381, Z -1.3333, A 0.000, B 0.000, C 0.000 }
gfCNCPoint1[17549] = {X 183.7431, Y 19.5458, Z -1.3333, A 0.000, B 0.000, C 0.000 }
gfCNCPoint1[17550] = {X 182.5380, Y 19.8868, Z -1.3333, A 0.000, B 0.000, C 0.000 }
gfCNCPoint1[17551] = {X 181.3956, Y 20.4002, Z -1.3333, A 0.000, B 0.000, C 0.000 }
gfCNCPoint1[17552] = {X 181.2442, Y 21.1598, Z -1.3333, A 0.000, B 0.000, C 0.000 }
gfCNCPoint1[17553] = {X 180.9619, Y 21.8810, Z -1.3333, A 0.000, B 0.000, C 0.000 }
gfCNCPoint1[17554] = {X 180.5575, Y 22.5416, Z -1.3333, A 0.000, B 0.000, C 0.000 }
gfCNCPoint1[17555] = {X 182.4466, Y 22.3528, Z -1.3333, A 0.000, B 0.000, C 0.000 }
gfCNCPoint1[17556] = {X 184.3414, Y 22.2348, Z -1.3333, A 0.000, B 0.000, C 0.000 }
gfCNCPoint1[17557] = {X 184.7766, Y 22.2190, Z -1.3333, A 0.000, B 0.000, C 0.000 }
gfCNCPoint1[17558] = {X 185.2118, Y 22.2014, Z -1.3333, A 0.000, B 0.000, C 0.000 }
gfCNCPoint1[17559] = {X 181.2193, Y 22.1012, Z -1.3333, A 0.000, B 0.000, C 0.000 }
gfCNCPoint1[17560] = {X 185.2152, Y 22.2813, Z -1.3333, A 0.000, B 0.000, C 0.000 }
gfCNCPoint1[17561] = {X 187.5451, Y 22.1587, Z -1.3333, A 0.000, B 0.000, C 0.000 }
gfCNCPoint1[17562] = {X 189.8719, Y 21.9879, Z -1.3333, A 0.000, B 0.000, C 0.000 }
gfCNCPoint1[17563] = {X 190.5075, Y 21.9068, Z -1.3333, A 0.000, B 0.000, C 0.000 }
gfCNCPoint1[17564] = {X 191.1268, Y 21.7427, Z -1.3333, A 0.000, B 0.000, C 0.000 }
gfCNCPoint1[17565] = {X 191.1533, Y 21.1789, Z -1.3333, A 0.000, B 0.000, C 0.000 }
gfCNCPoint1[17566] = {X 190.9478, Y 20.6533, Z -1.3333, A 0.000, B 0.000, C 0.000 }
gfCNCPoint1[17567] = {X 190.5460, Y 20.2569, Z -1.3333, A 0.000, B 0.000, C 0.000 }
gfCNCPoint1[17568] = {X 189.6782, Y 19.7912, Z -1.3333, A 0.000, B 0.000, C 0.000 }
gfCNCPoint1[17569] = {X 188.7497, Y 19.4628, Z -1.3333, A 0.000, B 0.000, C 0.000 }
gfCNCPoint1[17570] = {X 187.7821, Y 19.2793, Z -1.3333, A 0.000, B 0.000, C 0.000 }
gfCNCPoint1[17571] = {X 186.4269, Y 19.1955, Z -1.3333, A 0.000, B 0.000, C 0.000 }
gfCNCPoint1[17572] = {X 185.0705, Y 19.2583, Z -1.3333, A 0.000, B 0.000, C 0.000 }
gfCNCPoint1[17573] = {X 183.7289, Y 19.4670, Z -1.3333, A 0.000, B 0.000, C 0.000 }
gfCNCPoint1[17574] = {X 182.4923, Y 19.8183, Z -1.3333, A 0.000, B 0.000, C 0.000 }
gfCNCPoint1[17575] = {X 181.3216, Y 20.3494, Z -1.3333, A 0.000, B 0.000, C 0.000 }
gfCNCPoint1[17576] = {X 181.1582, Y 21.1710, Z -1.3333, A 0.000, B 0.000, C 0.000 }
gfCNCPoint1[17577] = {X 180.8393, Y 21.9455, Z -1.3333, A 0.000, B 0.000, C 0.000 }
gfCNCPoint1[17578] = {X 180.3770, Y 22.6440, Z -1.3333, A 0.000, B 0.000, C 0.000 }
gfCNCPoint1[17579] = {X 182.3566, Y 22.4405, Z -1.3333, A 0.000, B 0.000, C 0.000 }
gfCNCPoint1[17580] = {X 184.3427, Y 22.3148, Z -1.3333, A 0.000, B 0.000, C 0.000 }
gfCNCPoint1[17581] = {X 184.7790, Y 22.2989, Z -1.3333, A 0.000, B 0.000, C 0.000 }
gfCNCPoint1[17582] = {X 185.2152, Y 22.2813, Z -1.3333, A 0.000, B 0.000, C 0.000 }
gfCNCPoint1[17583] = {X 189.1817, Y 21.7649, Z -1.3333, A 0.000, B 0.000, C 0.000 }
gfCNCPoint1[17584] = {X 181.2227, Y 22.1811, Z -1.3333, A 0.000, B 0.000, C 0.000 }
gfCNCPoint1[17585] = {X 185.2186, Y 22.3613, Z -1.3333, A 0.000, B 0.000, C 0.000 }
gfCNCPoint1[17586] = {X 187.5497, Y 22.2386, Z -1.3333, A 0.000, B 0.000, C 0.000 }
gfCNCPoint1[17587] = {X 189.8777, Y 22.0677, Z -1.3333, A 0.000, B 0.000, C 0.000 }
gfCNCPoint1[17588] = {X 190.5441, Y 21.9811, Z -1.3333, A 0.000, B 0.000, C 0.000 }
gfCNCPoint1[17589] = {X 191.1925, Y 21.8048, Z -1.3333, A 0.000, B 0.000, C 0.000 }
gfCNCPoint1[17590] = {X 191.2503, Y 21.3480, Z -1.3333, A 0.000, B 0.000, C 0.000 }
gfCNCPoint1[17591] = {X 191.1605, Y 20.8964, Z -1.3333, A 0.000, B 0.000, C 0.000 }
gfCNCPoint1[17592] = {X 190.9322, Y 20.4965, Z -1.3333, A 0.000, B 0.000, C 0.000 }
gfCNCPoint1[17593] = {X 190.5891, Y 20.1895, Z -1.3333, A 0.000, B 0.000, C 0.000 }
gfCNCPoint1[17594] = {X 189.7105, Y 19.7181, Z -1.3333, A 0.000, B 0.000, C 0.000 }
gfCNCPoint1[17595] = {X 188.7705, Y 19.3856, Z -1.3333, A 0.000, B 0.000, C 0.000 }
gfCNCPoint1[17596] = {X 187.7910, Y 19.1998, Z -1.3333, A 0.000, B 0.000, C 0.000 }
gfCNCPoint1[17597] = {X 186.4273, Y 19.1155, Z -1.3333, A 0.000, B 0.000, C 0.000 }
gfCNCPoint1[17598] = {X 185.0624, Y 19.1787, Z -1.3333, A 0.000, B 0.000, C 0.000 }
gfCNCPoint1[17599] = {X 183.7123, Y 19.3887, Z -1.3333, A 0.000, B 0.000, C 0.000 }
gfCNCPoint1[17600] = {X 182.4466, Y 19.7499, Z -1.3333, A 0.000, B 0.000, C 0.000 }
gfCNCPoint1[17601] = {X 181.2497, Y 20.2976, Z -1.3333, A 0.000, B 0.000, C 0.000 }
gfCNCPoint1[17602] = {X 181.2398, Y 20.3518, Z -1.3333, A 0.000, B 0.000, C 0.000 }
gfCNCPoint1[17603] = {X 181.0789, Y 21.1544, Z -1.3333, A 0.000, B 0.000, C 0.000 }
gfCNCPoint1[17604] = {X 180.7666, Y 21.9110, Z -1.3333, A 0.000, B 0.000, C 0.000 }
gfCNCPoint1[17605] = {X 180.3148, Y 22.5937, Z -1.3333, A 0.000, B 0.000, C 0.000 }
gfCNCPoint1[17606] = {X 180.2501, Y 22.6716, Z -1.3333, A 0.000, B 0.000, C 0.000 }
gfCNCPoint1[17607] = {X 180.1835, Y 22.7479, Z -1.3333, A 0.000, B 0.000, C 0.000 }
gfCNCPoint1[17608] = {X 180.1890, Y 22.7481, Z -1.3333, A 0.000, B 0.000, C 0.000 }
gfCNCPoint1[17609] = {X 180.2878, Y 22.7357, Z -1.3333, A 0.000, B 0.000, C 0.000 }
gfCNCPoint1[17610] = {X 180.3867, Y 22.7234, Z -1.3333, A 0.000, B 0.000, C 0.000 }
gfCNCPoint1[17611] = {X 182.3630, Y 22.5202, Z -1.3333, A 0.000, B 0.000, C 0.000 }
gfCNCPoint1[17612] = {X 184.3458, Y 22.3948, Z -1.3333, A 0.000, B 0.000, C 0.000 }
gfCNCPoint1[17613] = {X 184.7822, Y 22.3789, Z -1.3333, A 0.000, B 0.000, C 0.000 }
gfCNCPoint1[17614] = {X 185.2186, Y 22.3613, Z -1.3333, A 0.000, B 0.000, C 0.000 }
gfCNCPoint1[17615] = {X 189.1851, Y 21.8448, Z -1.3333, A 0.000, B 0.000, C 0.000 }
gfCNCPoint1[17616] = {X 181.2260, Y 22.2611, Z -1.3333, A 0.000, B 0.000, C 0.000 }
gfCNCPoint1[17617] = {X 185.2220, Y 22.4412, Z -1.3333, A 0.000, B 0.000, C 0.000 }
gfCNCPoint1[17618] = {X 187.5542, Y 22.3185, Z -1.3333, A 0.000, B 0.000, C 0.000 }
gfCNCPoint1[17619] = {X 189.8835, Y 22.1475, Z -1.3333, A 0.000, B 0.000, C 0.000 }
gfCNCPoint1[17620] = {X 190.5801, Y 22.0555, Z -1.3333, A 0.000, B 0.000, C 0.000 }
gfCNCPoint1[17621] = {X 191.2570, Y 21.8669, Z -1.3333, A 0.000, B 0.000, C 0.000 }
gfCNCPoint1[17622] = {X 191.3310, Y 21.3762, Z -1.3333, A 0.000, B 0.000, C 0.000 }
gfCNCPoint1[17623] = {X 191.2425, Y 20.8878, Z -1.3333, A 0.000, B 0.000, C 0.000 }
gfCNCPoint1[17624] = {X 191.0009, Y 20.4543, Z -1.3333, A 0.000, B 0.000, C 0.000 }
gfCNCPoint1[17625] = {X 190.6322, Y 20.1221, Z -1.3333, A 0.000, B 0.000, C 0.000 }
gfCNCPoint1[17626] = {X 189.7429, Y 19.6449, Z -1.3333, A 0.000, B 0.000, C 0.000 }
gfCNCPoint1[17627] = {X 188.7914, Y 19.3084, Z -1.3333, A 0.000, B 0.000, C 0.000 }
gfCNCPoint1[17628] = {X 187.7998, Y 19.1203, Z -1.3333, A 0.000, B 0.000, C 0.000 }
gfCNCPoint1[17629] = {X 186.4276, Y 19.0355, Z -1.3333, A 0.000, B 0.000, C 0.000 }
gfCNCPoint1[17630] = {X 185.0543, Y 19.0991, Z -1.3333, A 0.000, B 0.000, C 0.000 }
gfCNCPoint1[17631] = {X 183.6958, Y 19.3105, Z -1.3333, A 0.000, B 0.000, C 0.000 }
gfCNCPoint1[17632] = {X 182.4008, Y 19.6815, Z -1.3333, A 0.000, B 0.000, C 0.000 }
gfCNCPoint1[17633] = {X 181.1777, Y 20.2461, Z -1.3333, A 0.000, B 0.000, C 0.000 }
gfCNCPoint1[17634] = {X 181.1606, Y 20.3406, Z -1.3333, A 0.000, B 0.000, C 0.000 }
gfCNCPoint1[17635] = {X 180.9651, Y 21.2476, Z -1.3333, A 0.000, B 0.000, C 0.000 }
gfCNCPoint1[17636] = {X 180.5734, Y 22.0888, Z -1.3333, A 0.000, B 0.000, C 0.000 }
gfCNCPoint1[17637] = {X 180.0050, Y 22.8222, Z -1.3333, A 0.000, B 0.000, C 0.000 }
gfCNCPoint1[17638] = {X 180.1927, Y 22.8283, Z -1.3333, A 0.000, B 0.000, C 0.000 }
gfCNCPoint1[17639] = {X 182.2672, Y 22.6085, Z -1.3333, A 0.000, B 0.000, C 0.000 }
gfCNCPoint1[17640] = {X 184.3489, Y 22.4747, Z -1.3333, A 0.000, B 0.000, C 0.000 }
gfCNCPoint1[17641] = {X 184.7855, Y 22.4588, Z -1.3333, A 0.000, B 0.000, C 0.000 }
gfCNCPoint1[17642] = {X 185.2220, Y 22.4412, Z -1.3333, A 0.000, B 0.000, C 0.000 }
gfCNCPoint1[17643] = {X 189.1885, Y 21.9247, Z -1.3333, A 0.000, B 0.000, C 0.000 }
gfCNCPoint1[17644] = {X 181.2294, Y 22.3410, Z -1.3333, A 0.000, B 0.000, C 0.000 }
gfCNCPoint1[17645] = {X 185.2253, Y 22.5211, Z -1.3333, A 0.000, B 0.000, C 0.000 }
gfCNCPoint1[17646] = {X 187.5588, Y 22.3983, Z -1.3333, A 0.000, B 0.000, C 0.000 }
gfCNCPoint1[17647] = {X 189.8893, Y 22.2272, Z -1.3333, A 0.000, B 0.000, C 0.000 }
gfCNCPoint1[17648] = {X 190.6156, Y 22.1299, Z -1.3333, A 0.000, B 0.000, C 0.000 }
gfCNCPoint1[17649] = {X 191.3204, Y 21.9291, Z -1.3333, A 0.000, B 0.000, C 0.000 }
gfCNCPoint1[17650] = {X 191.4112, Y 21.4046, Z -1.3333, A 0.000, B 0.000, C 0.000 }
gfCNCPoint1[17651] = {X 191.3244, Y 20.8795, Z -1.3333, A 0.000, B 0.000, C 0.000 }
gfCNCPoint1[17652] = {X 191.0696, Y 20.4122, Z -1.3333, A 0.000, B 0.000, C 0.000 }
gfCNCPoint1[17653] = {X 190.6753, Y 20.0547, Z -1.3333, A 0.000, B 0.000, C 0.000 }
gfCNCPoint1[17654] = {X 189.7752, Y 19.5717, Z -1.3333, A 0.000, B 0.000, C 0.000 }
gfCNCPoint1[17655] = {X 188.8123, Y 19.2311, Z -1.3333, A 0.000, B 0.000, C 0.000 }
gfCNCPoint1[17656] = {X 187.8087, Y 19.0408, Z -1.3333, A 0.000, B 0.000, C 0.000 }
gfCNCPoint1[17657] = {X 186.4280, Y 18.9555, Z -1.3333, A 0.000, B 0.000, C 0.000 }
gfCNCPoint1[17658] = {X 185.0461, Y 19.0195, Z -1.3333, A 0.000, B 0.000, C 0.000 }
gfCNCPoint1[17659] = {X 183.6792, Y 19.2322, Z -1.3333, A 0.000, B 0.000, C 0.000 }
gfCNCPoint1[17660] = {X 182.3550, Y 19.6132, Z -1.3333, A 0.000, B 0.000, C 0.000 }
gfCNCPoint1[17661] = {X 181.1058, Y 20.1947, Z -1.3333, A 0.000, B 0.000, C 0.000 }
gfCNCPoint1[17662] = {X 181.0813, Y 20.3294, Z -1.3333, A 0.000, B 0.000, C 0.000 }
gfCNCPoint1[17663] = {X 180.8699, Y 21.2785, Z -1.3333, A 0.000, B 0.000, C 0.000 }
gfCNCPoint1[17664] = {X 180.4399, Y 22.1505, Z -1.3333, A 0.000, B 0.000, C 0.000 }
gfCNCPoint1[17665] = {X 179.8158, Y 22.8961, Z -1.3333, A 0.000, B 0.000, C 0.000 }
gfCNCPoint1[17666] = {X 180.1965, Y 22.9084, Z -1.3333, A 0.000, B 0.000, C 0.000 }
gfCNCPoint1[17667] = {X 182.2706, Y 22.6885, Z -1.3333, A 0.000, B 0.000, C 0.000 }
gfCNCPoint1[17668] = {X 184.3521, Y 22.5546, Z -1.3333, A 0.000, B 0.000, C 0.000 }
gfCNCPoint1[17669] = {X 184.7887, Y 22.5387, Z -1.3333, A 0.000, B 0.000, C 0.000 }
gfCNCPoint1[17670] = {X 185.2253, Y 22.5211, Z -1.3333, A 0.000, B 0.000, C 0.000 }
gfCNCPoint1[17671] = {X 189.1919, Y 22.0047, Z -1.3333, A 0.000, B 0.000, C 0.000 }
gfCNCPoint1[17672] = {X 185.1537, Y 22.6042, Z -1.3333, A 0.000, B 0.000, C 0.000 }
gfCNCPoint1[17673] = {X 185.2287, Y 22.6011, Z -1.3333, A 0.000, B 0.000, C 0.000 }
gfCNCPoint1[17674] = {X 187.5634, Y 22.4782, Z -1.3333, A 0.000, B 0.000, C 0.000 }
gfCNCPoint1[17675] = {X 189.8950, Y 22.3070, Z -1.3333, A 0.000, B 0.000, C 0.000 }
gfCNCPoint1[17676] = {X 190.6506, Y 22.2042, Z -1.3333, A 0.000, B 0.000, C 0.000 }
gfCNCPoint1[17677] = {X 191.3828, Y 21.9913, Z -1.3333, A 0.000, B 0.000, C 0.000 }
gfCNCPoint1[17678] = {X 191.4908, Y 21.4334, Z -1.3333, A 0.000, B 0.000, C 0.000 }
gfCNCPoint1[17679] = {X 191.4061, Y 20.8714, Z -1.3333, A 0.000, B 0.000, C 0.000 }
gfCNCPoint1[17680] = {X 191.1383, Y 20.3702, Z -1.3333, A 0.000, B 0.000, C 0.000 }
gfCNCPoint1[17681] = {X 190.7183, Y 19.9873, Z -1.3333, A 0.000, B 0.000, C 0.000 }
gfCNCPoint1[17682] = {X 189.8076, Y 19.4986, Z -1.3333, A 0.000, B 0.000, C 0.000 }
gfCNCPoint1[17683] = {X 188.8331, Y 19.1539, Z -1.3333, A 0.000, B 0.000, C 0.000 }
gfCNCPoint1[17684] = {X 187.8176, Y 18.9612, Z -1.3333, A 0.000, B 0.000, C 0.000 }
gfCNCPoint1[17685] = {X 186.4284, Y 18.8755, Z -1.3333, A 0.000, B 0.000, C 0.000 }
gfCNCPoint1[17686] = {X 185.0380, Y 18.9400, Z -1.3333, A 0.000, B 0.000, C 0.000 }
gfCNCPoint1[17687] = {X 183.6627, Y 19.1539, Z -1.3333, A 0.000, B 0.000, C 0.000 }
gfCNCPoint1[17688] = {X 182.3092, Y 19.5450, Z -1.3333, A 0.000, B 0.000, C 0.000 }
gfCNCPoint1[17689] = {X 181.0337, Y 20.1436, Z -1.3333, A 0.000, B 0.000, C 0.000 }
gfCNCPoint1[17690] = {X 181.0020, Y 20.3183, Z -1.3333, A 0.000, B 0.000, C 0.000 }
gfCNCPoint1[17691] = {X 180.8538, Y 21.0695, Z -1.3333, A 0.000, B 0.000, C 0.000 }
gfCNCPoint1[17692] = {X 180.5651, Y 21.7787, Z -1.3333, A 0.000, B 0.000, C 0.000 }
gfCNCPoint1[17693] = {X 180.1466, Y 22.4199, Z -1.3333, A 0.000, B 0.000, C 0.000 }
gfCNCPoint1[17694] = {X 179.6136, Y 22.9696, Z -1.3333, A 0.000, B 0.000, C 0.000 }
gfCNCPoint1[17695] = {X 180.2003, Y 22.9886, Z -1.3333, A 0.000, B 0.000, C 0.000 }
gfCNCPoint1[17696] = {X 182.2741, Y 22.7685, Z -1.3333, A 0.000, B 0.000, C 0.000 }
gfCNCPoint1[17697] = {X 184.3552, Y 22.6346, Z -1.3333, A 0.000, B 0.000, C 0.000 }
gfCNCPoint1[17698] = {X 184.7920, Y 22.6187, Z -1.3333, A 0.000, B 0.000, C 0.000 }
gfCNCPoint1[17699] = {X 185.2287, Y 22.6011, Z -1.3333, A 0.000, B 0.000, C 0.000 }
gfCNCPoint1[17700] = {X 185.1443, Y 20.6028, Z -1.3333, A 0.000, B 0.000, C 0.000 }
gfCNCPoint1[17701] = {X 185.1443, Y 20.6028, Z 1.6667, A 0.000, B 0.000, C 0.000 }
gfCNCPoint1[17702] = {X 185.1443, Y 20.6028, Z 11.0000, A 0.000, B 0.000, C 0.000 }
gfCNCPoint1[17703] = {X 186.2322, Y 37.9131, Z 11.0000, A 0.000, B 0.000, C 0.000 }
gfCNCPoint1[17704] = {X 186.2322, Y 37.9131, Z 2.5000, A 0.000, B 0.000, C 0.000 }
gfCNCPoint1[17705] = {X 187.5941, Y 37.8330, Z 2.1345, A 0.000, B 0.000, C 0.000 }
gfCNCPoint1[17706] = {X 189.4252, Y 37.3846, Z 1.6293, A 0.000, B 0.000, C 0.000 }
gfCNCPoint1[17707] = {X 190.9864, Y 36.7119, Z 1.1738, A 0.000, B 0.000, C 0.000 }
gfCNCPoint1[17708] = {X 191.6937, Y 36.3238, Z 0.9576, A 0.000, B 0.000, C 0.000 }
gfCNCPoint1[17709] = {X 192.4466, Y 35.8120, Z 0.7137, A 0.000, B 0.000, C 0.000 }
gfCNCPoint1[17710] = {X 192.4699, Y 35.2979, Z 0.5758, A 0.000, B 0.000, C 0.000 }
gfCNCPoint1[17711] = {X 192.6319, Y 34.6331, Z 0.3924, A 0.000, B 0.000, C 0.000 }
gfCNCPoint1[17712] = {X 192.8477, Y 34.1658, Z 0.2545, A 0.000, B 0.000, C 0.000 }
gfCNCPoint1[17713] = {X 192.7390, Y 34.1912, Z 0.2246, A 0.000, B 0.000, C 0.000 }
gfCNCPoint1[17714] = {X 191.4117, Y 34.4412, Z -0.1373, A 0.000, B 0.000, C 0.000 }
gfCNCPoint1[17715] = {X 190.5778, Y 34.5485, Z -0.3626, A 0.000, B 0.000, C 0.000 }
gfCNCPoint1[17716] = {X 189.2271, Y 34.6429, Z -0.7254, A 0.000, B 0.000, C 0.000 }
gfCNCPoint1[17717] = {X 186.9624, Y 34.7819, Z -1.3333, A 0.000, B 0.000, C 0.000 }
gfCNCPoint1[17718] = {X 182.5786, Y 35.0511, Z -1.3333, A 0.000, B 0.000, C 0.000 }
gfCNCPoint1[17719] = {X 181.8183, Y 35.1388, Z -1.3333, A 0.000, B 0.000, C 0.000 }
gfCNCPoint1[17720] = {X 181.0717, Y 35.3071, Z -1.3333, A 0.000, B 0.000, C 0.000 }
gfCNCPoint1[17721] = {X 181.0635, Y 35.3817, Z -1.3333, A 0.000, B 0.000, C 0.000 }
gfCNCPoint1[17722] = {X 181.0634, Y 35.4566, Z -1.3333, A 0.000, B 0.000, C 0.000 }
gfCNCPoint1[17723] = {X 181.1562, Y 35.9991, Z -1.3333, A 0.000, B 0.000, C 0.000 }
gfCNCPoint1[17724] = {X 181.4128, Y 36.4860, Z -1.3333, A 0.000, B 0.000, C 0.000 }
gfCNCPoint1[17725] = {X 181.8077, Y 36.8693, Z -1.3333, A 0.000, B 0.000, C 0.000 }
gfCNCPoint1[17726] = {X 182.4210, Y 37.2302, Z -1.3333, A 0.000, B 0.000, C 0.000 }
gfCNCPoint1[17727] = {X 183.0843, Y 37.4876, Z -1.3333, A 0.000, B 0.000, C 0.000 }
gfCNCPoint1[17728] = {X 184.4931, Y 37.8023, Z -1.3333, A 0.000, B 0.000, C 0.000 }
gfCNCPoint1[17729] = {X 185.9319, Y 37.9183, Z -1.3333, A 0.000, B 0.000, C 0.000 }
gfCNCPoint1[17730] = {X 187.3728, Y 37.8336, Z -1.3333, A 0.000, B 0.000, C 0.000 }
gfCNCPoint1[17731] = {X 188.7881, Y 37.5497, Z -1.3333, A 0.000, B 0.000, C 0.000 }
gfCNCPoint1[17732] = {X 190.1503, Y 37.0722, Z -1.3333, A 0.000, B 0.000, C 0.000 }
gfCNCPoint1[17733] = {X 191.3284, Y 36.4967, Z -1.3333, A 0.000, B 0.000, C 0.000 }
gfCNCPoint1[17734] = {X 192.4466, Y 35.8120, Z -1.3333, A 0.000, B 0.000, C 0.000 }
gfCNCPoint1[17735] = {X 192.5672, Y 34.9695, Z -1.3333, A 0.000, B 0.000, C 0.000 }
gfCNCPoint1[17736] = {X 192.8477, Y 34.1658, Z -1.3333, A 0.000, B 0.000, C 0.000 }
gfCNCPoint1[17737] = {X 192.7390, Y 34.1912, Z -1.3333, A 0.000, B 0.000, C 0.000 }
gfCNCPoint1[17738] = {X 190.9896, Y 34.4682, Z -1.3333, A 0.000, B 0.000, C 0.000 }
gfCNCPoint1[17739] = {X 189.2271, Y 34.6429, Z -1.3333, A 0.000, B 0.000, C 0.000 }
gfCNCPoint1[17740] = {X 186.9624, Y 34.7819, Z -1.3333, A 0.000, B 0.000, C 0.000 }
gfCNCPoint1[17741] = {X 190.9561, Y 34.8058, Z -1.3333, A 0.000, B 0.000, C 0.000 }
gfCNCPoint1[17742] = {X 186.9575, Y 34.7021, Z -1.3333, A 0.000, B 0.000, C 0.000 }
gfCNCPoint1[17743] = {X 182.5737, Y 34.9712, Z -1.3333, A 0.000, B 0.000, C 0.000 }
gfCNCPoint1[17744] = {X 181.7808, Y 35.0641, Z -1.3333, A 0.000, B 0.000, C 0.000 }
gfCNCPoint1[17745] = {X 181.0028, Y 35.2436, Z -1.3333, A 0.000, B 0.000, C 0.000 }
gfCNCPoint1[17746] = {X 180.9859, Y 35.3477, Z -1.3333, A 0.000, B 0.000, C 0.000 }
gfCNCPoint1[17747] = {X 180.9834, Y 35.4531, Z -1.3333, A 0.000, B 0.000, C 0.000 }
gfCNCPoint1[17748] = {X 181.0795, Y 36.0220, Z -1.3333, A 0.000, B 0.000, C 0.000 }
gfCNCPoint1[17749] = {X 181.3478, Y 36.5328, Z -1.3333, A 0.000, B 0.000, C 0.000 }
gfCNCPoint1[17750] = {X 181.7617, Y 36.9348, Z -1.3333, A 0.000, B 0.000, C 0.000 }
gfCNCPoint1[17751] = {X 182.3861, Y 37.3022, Z -1.3333, A 0.000, B 0.000, C 0.000 }
gfCNCPoint1[17752] = {X 183.0615, Y 37.5643, Z -1.3333, A 0.000, B 0.000, C 0.000 }
gfCNCPoint1[17753] = {X 184.4811, Y 37.8814, Z -1.3333, A 0.000, B 0.000, C 0.000 }
gfCNCPoint1[17754] = {X 185.9310, Y 37.9983, Z -1.3333, A 0.000, B 0.000, C 0.000 }
gfCNCPoint1[17755] = {X 187.3831, Y 37.9130, Z -1.3333, A 0.000, B 0.000, C 0.000 }
gfCNCPoint1[17756] = {X 188.8093, Y 37.6269, Z -1.3333, A 0.000, B 0.000, C 0.000 }
gfCNCPoint1[17757] = {X 190.1819, Y 37.1456, Z -1.3333, A 0.000, B 0.000, C 0.000 }
gfCNCPoint1[17758] = {X 191.3846, Y 36.5571, Z -1.3333, A 0.000, B 0.000, C 0.000 }
gfCNCPoint1[17759] = {X 192.5249, Y 35.8555, Z -1.3333, A 0.000, B 0.000, C 0.000 }
gfCNCPoint1[17760] = {X 192.6604, Y 34.9267, Z -1.3333, A 0.000, B 0.000, C 0.000 }
gfCNCPoint1[17761] = {X 192.9933, Y 34.0491, Z -1.3333, A 0.000, B 0.000, C 0.000 }
gfCNCPoint1[17762] = {X 192.7316, Y 34.1112, Z -1.3333, A 0.000, B 0.000, C 0.000 }
gfCNCPoint1[17763] = {X 190.9841, Y 34.3883, Z -1.3333, A 0.000, B 0.000, C 0.000 }
gfCNCPoint1[17764] = {X 189.2235, Y 34.5629, Z -1.3333, A 0.000, B 0.000, C 0.000 }
gfCNCPoint1[17765] = {X 186.9575, Y 34.7021, Z -1.3333, A 0.000, B 0.000, C 0.000 }
gfCNCPoint1[17766] = {X 183.0016, Y 35.2942, Z -1.3333, A 0.000, B 0.000, C 0.000 }
gfCNCPoint1[17767] = {X 190.9512, Y 34.7260, Z -1.3333, A 0.000, B 0.000, C 0.000 }
gfCNCPoint1[17768] = {X 186.9526, Y 34.6222, Z -1.3333, A 0.000, B 0.000, C 0.000 }
gfCNCPoint1[17769] = {X 182.5688, Y 34.8914, Z -1.3333, A 0.000, B 0.000, C 0.000 }
gfCNCPoint1[17770] = {X 181.7448, Y 34.9891, Z -1.3333, A 0.000, B 0.000, C 0.000 }
gfCNCPoint1[17771] = {X 180.9370, Y 35.1796, Z -1.3333, A 0.000, B 0.000, C 0.000 }
gfCNCPoint1[17772] = {X 180.9089, Y 35.3160, Z -1.3333, A 0.000, B 0.000, C 0.000 }
gfCNCPoint1[17773] = {X 180.9034, Y 35.4552, Z -1.3333, A 0.000, B 0.000, C 0.000 }
gfCNCPoint1[17774] = {X 181.0040, Y 36.0484, Z -1.3333, A 0.000, B 0.000, C 0.000 }
gfCNCPoint1[17775] = {X 181.2840, Y 36.5810, Z -1.3333, A 0.000, B 0.000, C 0.000 }
gfCNCPoint1[17776] = {X 181.7157, Y 37.0002, Z -1.3333, A 0.000, B 0.000, C 0.000 }
gfCNCPoint1[17777] = {X 182.3513, Y 37.3742, Z -1.3333, A 0.000, B 0.000, C 0.000 }
gfCNCPoint1[17778] = {X 183.0387, Y 37.6410, Z -1.3333, A 0.000, B 0.000, C 0.000 }
gfCNCPoint1[17779] = {X 184.4692, Y 37.9605, Z -1.3333, A 0.000, B 0.000, C 0.000 }
gfCNCPoint1[17780] = {X 185.9301, Y 38.0783, Z -1.3333, A 0.000, B 0.000, C 0.000 }
gfCNCPoint1[17781] = {X 187.3933, Y 37.9923, Z -1.3333, A 0.000, B 0.000, C 0.000 }
gfCNCPoint1[17782] = {X 188.8304, Y 37.7040, Z -1.3333, A 0.000, B 0.000, C 0.000 }
gfCNCPoint1[17783] = {X 190.2136, Y 37.2191, Z -1.3333, A 0.000, B 0.000, C 0.000 }
gfCNCPoint1[17784] = {X 191.4410, Y 36.6174, Z -1.3333, A 0.000, B 0.000, C 0.000 }
gfCNCPoint1[17785] = {X 192.6036, Y 35.8985, Z -1.3333, A 0.000, B 0.000, C 0.000 }
gfCNCPoint1[17786] = {X 192.6774, Y 35.2158, Z -1.3333, A 0.000, B 0.000, C 0.000 }
gfCNCPoint1[17787] = {X 192.8604, Y 34.5539, Z -1.3333, A 0.000, B 0.000, C 0.000 }
gfCNCPoint1[17788] = {X 193.1478, Y 33.9303, Z -1.3333, A 0.000, B 0.000, C 0.000 }
gfCNCPoint1[17789] = {X 192.7149, Y 34.0329, Z -1.3333, A 0.000, B 0.000, C 0.000 }
gfCNCPoint1[17790] = {X 190.9732, Y 34.3090, Z -1.3333, A 0.000, B 0.000, C 0.000 }
gfCNCPoint1[17791] = {X 189.2183, Y 34.4831, Z -1.3333, A 0.000, B 0.000, C 0.000 }
gfCNCPoint1[17792] = {X 186.9526, Y 34.6222, Z -1.3333, A 0.000, B 0.000, C 0.000 }
gfCNCPoint1[17793] = {X 182.9967, Y 35.2144, Z -1.3333, A 0.000, B 0.000, C 0.000 }
gfCNCPoint1[17794] = {X 190.9463, Y 34.6461, Z -1.3333, A 0.000, B 0.000, C 0.000 }
gfCNCPoint1[17795] = {X 186.9477, Y 34.5424, Z -1.3333, A 0.000, B 0.000, C 0.000 }
gfCNCPoint1[17796] = {X 182.5639, Y 34.8115, Z -1.3333, A 0.000, B 0.000, C 0.000 }
gfCNCPoint1[17797] = {X 181.7100, Y 34.9141, Z -1.3333, A 0.000, B 0.000, C 0.000 }
gfCNCPoint1[17798] = {X 180.8737, Y 35.1150, Z -1.3333, A 0.000, B 0.000, C 0.000 }
gfCNCPoint1[17799] = {X 180.8325, Y 35.2838, Z -1.3333, A 0.000, B 0.000, C 0.000 }
gfCNCPoint1[17800] = {X 180.8234, Y 35.4572, Z -1.3333, A 0.000, B 0.000, C 0.000 }
gfCNCPoint1[17801] = {X 180.9285, Y 36.0749, Z -1.3333, A 0.000, B 0.000, C 0.000 }
gfCNCPoint1[17802] = {X 181.2202, Y 36.6293, Z -1.3333, A 0.000, B 0.000, C 0.000 }
gfCNCPoint1[17803] = {X 181.6697, Y 37.0657, Z -1.3333, A 0.000, B 0.000, C 0.000 }
gfCNCPoint1[17804] = {X 182.3164, Y 37.4462, Z -1.3333, A 0.000, B 0.000, C 0.000 }
gfCNCPoint1[17805] = {X 183.0159, Y 37.7176, Z -1.3333, A 0.000, B 0.000, C 0.000 }
gfCNCPoint1[17806] = {X 184.4572, Y 38.0396, Z -1.3333, A 0.000, B 0.000, C 0.000 }
gfCNCPoint1[17807] = {X 185.9293, Y 38.1583, Z -1.3333, A 0.000, B 0.000, C 0.000 }
gfCNCPoint1[17808] = {X 187.4036, Y 38.0716, Z -1.3333, A 0.000, B 0.000, C 0.000 }
gfCNCPoint1[17809] = {X 188.8516, Y 37.7812, Z -1.3333, A 0.000, B 0.000, C 0.000 }
gfCNCPoint1[17810] = {X 190.2453, Y 37.2926, Z -1.3333, A 0.000, B 0.000, C 0.000 }
gfCNCPoint1[17811] = {X 191.4976, Y 36.6775, Z -1.3333, A 0.000, B 0.000, C 0.000 }
gfCNCPoint1[17812] = {X 192.6827, Y 35.9411, Z -1.3333, A 0.000, B 0.000, C 0.000 }
gfCNCPoint1[17813] = {X 192.7627, Y 35.1962, Z -1.3333, A 0.000, B 0.000, C 0.000 }
gfCNCPoint1[17814] = {X 192.9750, Y 34.4777, Z -1.3333, A 0.000, B 0.000, C 0.000 }
gfCNCPoint1[17815] = {X 193.3128, Y 33.8089, Z -1.3333, A 0.000, B 0.000, C 0.000 }
gfCNCPoint1[17816] = {X 192.6983, Y 33.9546, Z -1.3333, A 0.000, B 0.000, C 0.000 }
gfCNCPoint1[17817] = {X 190.9622, Y 34.2298, Z -1.3333, A 0.000, B 0.000, C 0.000 }
gfCNCPoint1[17818] = {X 189.2130, Y 34.4033, Z -1.3333, A 0.000, B 0.000, C 0.000 }
gfCNCPoint1[17819] = {X 186.9477, Y 34.5424, Z -1.3333, A 0.000, B 0.000, C 0.000 }
gfCNCPoint1[17820] = {X 182.9918, Y 35.1346, Z -1.3333, A 0.000, B 0.000, C 0.000 }
gfCNCPoint1[17821] = {X 190.9414, Y 34.5663, Z -1.3333, A 0.000, B 0.000, C 0.000 }
gfCNCPoint1[17822] = {X 186.9428, Y 34.4625, Z -1.3333, A 0.000, B 0.000, C 0.000 }
gfCNCPoint1[17823] = {X 182.5590, Y 34.7317, Z -1.3333, A 0.000, B 0.000, C 0.000 }
gfCNCPoint1[17824] = {X 181.6762, Y 34.8389, Z -1.3333, A 0.000, B 0.000, C 0.000 }
gfCNCPoint1[17825] = {X 180.8124, Y 35.0501, Z -1.3333, A 0.000, B 0.000, C 0.000 }
gfCNCPoint1[17826] = {X 180.7567, Y 35.2511, Z -1.3333, A 0.000, B 0.000, C 0.000 }
gfCNCPoint1[17827] = {X 180.7434, Y 35.4593, Z -1.3333, A 0.000, B 0.000, C 0.000 }
gfCNCPoint1[17828] = {X 180.8530, Y 36.1013, Z -1.3333, A 0.000, B 0.000, C 0.000 }
gfCNCPoint1[17829] = {X 181.1564, Y 36.6775, Z -1.3333, A 0.000, B 0.000, C 0.000 }
gfCNCPoint1[17830] = {X 181.6237, Y 37.1311, Z -1.3333, A 0.000, B 0.000, C 0.000 }
gfCNCPoint1[17831] = {X 182.2815, Y 37.5182, Z -1.3333, A 0.000, B 0.000, C 0.000 }
gfCNCPoint1[17832] = {X 182.9930, Y 37.7943, Z -1.3333, A 0.000, B 0.000, C 0.000 }
gfCNCPoint1[17833] = {X 184.4452, Y 38.1187, Z -1.3333, A 0.000, B 0.000, C 0.000 }
gfCNCPoint1[17834] = {X 185.9284, Y 38.2383, Z -1.3333, A 0.000, B 0.000, C 0.000 }
gfCNCPoint1[17835] = {X 187.4138, Y 38.1510, Z -1.3333, A 0.000, B 0.000, C 0.000 }
gfCNCPoint1[17836] = {X 188.8727, Y 37.8583, Z -1.3333, A 0.000, B 0.000, C 0.000 }
gfCNCPoint1[17837] = {X 190.2769, Y 37.3660, Z -1.3333, A 0.000, B 0.000, C 0.000 }
gfCNCPoint1[17838] = {X 191.5545, Y 36.7374, Z -1.3333, A 0.000, B 0.000, C 0.000 }
gfCNCPoint1[17839] = {X 192.7622, Y 35.9833, Z -1.3333, A 0.000, B 0.000, C 0.000 }
gfCNCPoint1[17840] = {X 192.8359, Y 35.2386, Z -1.3333, A 0.000, B 0.000, C 0.000 }
gfCNCPoint1[17841] = {X 193.0444, Y 34.5198, Z -1.3333, A 0.000, B 0.000, C 0.000 }
gfCNCPoint1[17842] = {X 193.3806, Y 33.8513, Z -1.3333, A 0.000, B 0.000, C 0.000 }
gfCNCPoint1[17843] = {X 193.4234, Y 33.7841, Z -1.3333, A 0.000, B 0.000, C 0.000 }
gfCNCPoint1[17844] = {X 193.4675, Y 33.7179, Z -1.3333, A 0.000, B 0.000, C 0.000 }
gfCNCPoint1[17845] = {X 193.3654, Y 33.7142, Z -1.3333, A 0.000, B 0.000, C 0.000 }
gfCNCPoint1[17846] = {X 192.6816, Y 33.8764, Z -1.3333, A 0.000, B 0.000, C 0.000 }
gfCNCPoint1[17847] = {X 190.9512, Y 34.1505, Z -1.3333, A 0.000, B 0.000, C 0.000 }
gfCNCPoint1[17848] = {X 189.2078, Y 34.3235, Z -1.3333, A 0.000, B 0.000, C 0.000 }
gfCNCPoint1[17849] = {X 186.9428, Y 34.4625, Z -1.3333, A 0.000, B 0.000, C 0.000 }
gfCNCPoint1[17850] = {X 182.9869, Y 35.0547, Z -1.3333, A 0.000, B 0.000, C 0.000 }
gfCNCPoint1[17851] = {X 190.9365, Y 34.4864, Z -1.3333, A 0.000, B 0.000, C 0.000 }
gfCNCPoint1[17852] = {X 186.9379, Y 34.3827, Z -1.3333, A 0.000, B 0.000, C 0.000 }
gfCNCPoint1[17853] = {X 182.5541, Y 34.6518, Z -1.3333, A 0.000, B 0.000, C 0.000 }
gfCNCPoint1[17854] = {X 181.6433, Y 34.7636, Z -1.3333, A 0.000, B 0.000, C 0.000 }
gfCNCPoint1[17855] = {X 180.7528, Y 34.9849, Z -1.3333, A 0.000, B 0.000, C 0.000 }
gfCNCPoint1[17856] = {X 180.6813, Y 35.2181, Z -1.3333, A 0.000, B 0.000, C 0.000 }
gfCNCPoint1[17857] = {X 180.6635, Y 35.4613, Z -1.3333, A 0.000, B 0.000, C 0.000 }
gfCNCPoint1[17858] = {X 180.7775, Y 36.1277, Z -1.3333, A 0.000, B 0.000, C 0.000 }
gfCNCPoint1[17859] = {X 181.0926, Y 36.7258, Z -1.3333, A 0.000, B 0.000, C 0.000 }
gfCNCPoint1[17860] = {X 181.5777, Y 37.1966, Z -1.3333, A 0.000, B 0.000, C 0.000 }
gfCNCPoint1[17861] = {X 182.2467, Y 37.5902, Z -1.3333, A 0.000, B 0.000, C 0.000 }
gfCNCPoint1[17862] = {X 182.9702, Y 37.8710, Z -1.3333, A 0.000, B 0.000, C 0.000 }
gfCNCPoint1[17863] = {X 184.4333, Y 38.1978, Z -1.3333, A 0.000, B 0.000, C 0.000 }
gfCNCPoint1[17864] = {X 185.9275, Y 38.3183, Z -1.3333, A 0.000, B 0.000, C 0.000 }
gfCNCPoint1[17865] = {X 187.4240, Y 38.2303, Z -1.3333, A 0.000, B 0.000, C 0.000 }
gfCNCPoint1[17866] = {X 188.8939, Y 37.9355, Z -1.3333, A 0.000, B 0.000, C 0.000 }
gfCNCPoint1[17867] = {X 190.3086, Y 37.4395, Z -1.3333, A 0.000, B 0.000, C 0.000 }
gfCNCPoint1[17868] = {X 191.6116, Y 36.7972, Z -1.3333, A 0.000, B 0.000, C 0.000 }
gfCNCPoint1[17869] = {X 192.8422, Y 36.0250, Z -1.3333, A 0.000, B 0.000, C 0.000 }
gfCNCPoint1[17870] = {X 192.9290, Y 35.1818, Z -1.3333, A 0.000, B 0.000, C 0.000 }
gfCNCPoint1[17871] = {X 193.1917, Y 34.3757, Z -1.3333, A 0.000, B 0.000, C 0.000 }
gfCNCPoint1[17872] = {X 193.6183, Y 33.6431, Z -1.3333, A 0.000, B 0.000, C 0.000 }
gfCNCPoint1[17873] = {X 193.3575, Y 33.6339, Z -1.3333, A 0.000, B 0.000, C 0.000 }
gfCNCPoint1[17874] = {X 192.6650, Y 33.7981, Z -1.3333, A 0.000, B 0.000, C 0.000 }
gfCNCPoint1[17875] = {X 190.9403, Y 34.0713, Z -1.3333, A 0.000, B 0.000, C 0.000 }
gfCNCPoint1[17876] = {X 189.2026, Y 34.2436, Z -1.3333, A 0.000, B 0.000, C 0.000 }
gfCNCPoint1[17877] = {X 186.9379, Y 34.3827, Z -1.3333, A 0.000, B 0.000, C 0.000 }
gfCNCPoint1[17878] = {X 182.9820, Y 34.9749, Z -1.3333, A 0.000, B 0.000, C 0.000 }
gfCNCPoint1[17879] = {X 182.9820, Y 34.9749, Z 1.6667, A 0.000, B 0.000, C 0.000 }
gfCNCPoint1[17880] = {X 182.9820, Y 34.9749, Z 11.0000, A 0.000, B 0.000, C 0.000 }
gfCNCPoint1[17881] = {X 165.6772, Y 73.8165, Z 11.0000, A 0.000, B 0.000, C 0.000 }
gfCNCPoint1[17882] = {X 165.6772, Y 73.8165, Z 2.5000, A 0.000, B 0.000, C 0.000 }
gfCNCPoint1[17883] = {X 161.3996, Y 78.5670, Z 0.7871, A 0.000, B 0.000, C 0.000 }
gfCNCPoint1[17884] = {X 169.3132, Y 78.5670, Z -1.3333, A 0.000, B 0.000, C 0.000 }
gfCNCPoint1[17885] = {X 169.3132, Y 76.1670, Z -1.3333, A 0.000, B 0.000, C 0.000 }
gfCNCPoint1[17886] = {X 171.8361, Y 76.1670, Z -1.3333, A 0.000, B 0.000, C 0.000 }
gfCNCPoint1[17887] = {X 169.3147, Y 73.3634, Z -1.3333, A 0.000, B 0.000, C 0.000 }
gfCNCPoint1[17888] = {X 166.7903, Y 76.1670, Z -1.3333, A 0.000, B 0.000, C 0.000 }
gfCNCPoint1[17889] = {X 169.3132, Y 76.1670, Z -1.3333, A 0.000, B 0.000, C 0.000 }
gfCNCPoint1[17890] = {X 169.3132, Y 78.5670, Z -1.3333, A 0.000, B 0.000, C 0.000 }
gfCNCPoint1[17891] = {X 177.2224, Y 78.5670, Z -1.3333, A 0.000, B 0.000, C 0.000 }
gfCNCPoint1[17892] = {X 169.3158, Y 69.7756, Z -1.3333, A 0.000, B 0.000, C 0.000 }
gfCNCPoint1[17893] = {X 161.3996, Y 78.5670, Z -1.3333, A 0.000, B 0.000, C 0.000 }
gfCNCPoint1[17894] = {X 169.3132, Y 78.5670, Z -1.3333, A 0.000, B 0.000, C 0.000 }
gfCNCPoint1[17895] = {X 169.3132, Y 74.6470, Z -1.3333, A 0.000, B 0.000, C 0.000 }
gfCNCPoint1[17896] = {X 169.3132, Y 78.6470, Z -1.3333, A 0.000, B 0.000, C 0.000 }
gfCNCPoint1[17897] = {X 177.4019, Y 78.6470, Z -1.3333, A 0.000, B 0.000, C 0.000 }
gfCNCPoint1[17898] = {X 169.3159, Y 69.6560, Z -1.3333, A 0.000, B 0.000, C 0.000 }
gfCNCPoint1[17899] = {X 161.2199, Y 78.6470, Z -1.3333, A 0.000, B 0.000, C 0.000 }
gfCNCPoint1[17900] = {X 169.3132, Y 78.6470, Z -1.3333, A 0.000, B 0.000, C 0.000 }
gfCNCPoint1[17901] = {X 169.3132, Y 74.6470, Z -1.3333, A 0.000, B 0.000, C 0.000 }
gfCNCPoint1[17902] = {X 169.3132, Y 74.7270, Z -1.3333, A 0.000, B 0.000, C 0.000 }
gfCNCPoint1[17903] = {X 169.3132, Y 78.7270, Z -1.3333, A 0.000, B 0.000, C 0.000 }
gfCNCPoint1[17904] = {X 177.5814, Y 78.7270, Z -1.3333, A 0.000, B 0.000, C 0.000 }
gfCNCPoint1[17905] = {X 169.3159, Y 69.5364, Z -1.3333, A 0.000, B 0.000, C 0.000 }
gfCNCPoint1[17906] = {X 161.0403, Y 78.7270, Z -1.3333, A 0.000, B 0.000, C 0.000 }
gfCNCPoint1[17907] = {X 169.3132, Y 78.7270, Z -1.3333, A 0.000, B 0.000, C 0.000 }
gfCNCPoint1[17908] = {X 169.3132, Y 74.7270, Z -1.3333, A 0.000, B 0.000, C 0.000 }
gfCNCPoint1[17909] = {X 169.3132, Y 74.8070, Z -1.3333, A 0.000, B 0.000, C 0.000 }
gfCNCPoint1[17910] = {X 169.3132, Y 78.8070, Z -1.3333, A 0.000, B 0.000, C 0.000 }
gfCNCPoint1[17911] = {X 177.7610, Y 78.8070, Z -1.3333, A 0.000, B 0.000, C 0.000 }
gfCNCPoint1[17912] = {X 169.3159, Y 69.4168, Z -1.3333, A 0.000, B 0.000, C 0.000 }
gfCNCPoint1[17913] = {X 160.8606, Y 78.8070, Z -1.3333, A 0.000, B 0.000, C 0.000 }
gfCNCPoint1[17914] = {X 169.3132, Y 78.8070, Z -1.3333, A 0.000, B 0.000, C 0.000 }
gfCNCPoint1[17915] = {X 169.3132, Y 74.8070, Z -1.3333, A 0.000, B 0.000, C 0.000 }
gfCNCPoint1[17916] = {X 169.3132, Y 74.8870, Z -1.3333, A 0.000, B 0.000, C 0.000 }
gfCNCPoint1[17917] = {X 169.3132, Y 78.8870, Z -1.3333, A 0.000, B 0.000, C 0.000 }
gfCNCPoint1[17918] = {X 177.9405, Y 78.8870, Z -1.3333, A 0.000, B 0.000, C 0.000 }
gfCNCPoint1[17919] = {X 169.3160, Y 69.2972, Z -1.3333, A 0.000, B 0.000, C 0.000 }
gfCNCPoint1[17920] = {X 160.6809, Y 78.8870, Z -1.3333, A 0.000, B 0.000, C 0.000 }
gfCNCPoint1[17921] = {X 169.3132, Y 78.8870, Z -1.3333, A 0.000, B 0.000, C 0.000 }
gfCNCPoint1[17922] = {X 169.3132, Y 74.8870, Z -1.3333, A 0.000, B 0.000, C 0.000 }
gfCNCPoint1[17923] = {X 169.3132, Y 74.9670, Z -1.3333, A 0.000, B 0.000, C 0.000 }
gfCNCPoint1[17924] = {X 169.3132, Y 78.9670, Z -1.3333, A 0.000, B 0.000, C 0.000 }
gfCNCPoint1[17925] = {X 178.1201, Y 78.9670, Z -1.3333, A 0.000, B 0.000, C 0.000 }
gfCNCPoint1[17926] = {X 169.3160, Y 69.1776, Z -1.3333, A 0.000, B 0.000, C 0.000 }
gfCNCPoint1[17927] = {X 160.5012, Y 78.9670, Z -1.3333, A 0.000, B 0.000, C 0.000 }
gfCNCPoint1[17928] = {X 169.3132, Y 78.9670, Z -1.3333, A 0.000, B 0.000, C 0.000 }
gfCNCPoint1[17929] = {X 169.3132, Y 74.9670, Z -1.3333, A 0.000, B 0.000, C 0.000 }
gfCNCPoint1[17930] = {X 169.3132, Y 74.9670, Z 1.6667, A 0.000, B 0.000, C 0.000 }
gfCNCPoint1[17931] = {X 169.3132, Y 74.9670, Z 11.0000, A 0.000, B 0.000, C 0.000 }
gfCNCPoint1[17932] = {X 11.7116, Y 37.8802, Z 11.0000, A 0.000, B 0.000, C 0.000 }
gfCNCPoint1[17933] = {X 11.7116, Y 37.8802, Z 2.5000, A 0.000, B 0.000, C 0.000 }
gfCNCPoint1[17934] = {X 12.5002, Y 37.9520, Z 2.2878, A 0.000, B 0.000, C 0.000 }
gfCNCPoint1[17935] = {X 14.1409, Y 37.8407, Z 1.8472, A 0.000, B 0.000, C 0.000 }
gfCNCPoint1[17936] = {X 15.7434, Y 37.4719, Z 1.4066, A 0.000, B 0.000, C 0.000 }
gfCNCPoint1[17937] = {X 17.3070, Y 36.8446, Z 0.9552, A 0.000, B 0.000, C 0.000 }
gfCNCPoint1[17938] = {X 18.2945, Y 36.3176, Z 0.6552, A 0.000, B 0.000, C 0.000 }
gfCNCPoint1[17939] = {X 19.0345, Y 35.8124, Z 0.4152, A 0.000, B 0.000, C 0.000 }
gfCNCPoint1[17940] = {X 19.0577, Y 35.2983, Z 0.2772, A 0.000, B 0.000, C 0.000 }
gfCNCPoint1[17941] = {X 19.2193, Y 34.6345, Z 0.0942, A 0.000, B 0.000, C 0.000 }
gfCNCPoint1[17942] = {X 19.4349, Y 34.1672, Z -0.0437, A 0.000, B 0.000, C 0.000 }
gfCNCPoint1[17943] = {X 18.1955, Y 34.4158, Z -0.3824, A 0.000, B 0.000, C 0.000 }
gfCNCPoint1[17944] = {X 17.3716, Y 34.5275, Z -0.6052, A 0.000, B 0.000, C 0.000 }
gfCNCPoint1[17945] = {X 16.1107, Y 34.6182, Z -0.9439, A 0.000, B 0.000, C 0.000 }
gfCNCPoint1[17946] = {X 15.3861, Y 34.6720, Z -1.1386, A 0.000, B 0.000, C 0.000 }
gfCNCPoint1[17947] = {X 14.6611, Y 34.7215, Z -1.3333, A 0.000, B 0.000, C 0.000 }
gfCNCPoint1[17948] = {X 12.2609, Y 34.8741, Z -1.3333, A 0.000, B 0.000, C 0.000 }
gfCNCPoint1[17949] = {X 9.8594, Y 35.0039, Z -1.3333, A 0.000, B 0.000, C 0.000 }
gfCNCPoint1[17950] = {X 8.7531, Y 35.0944, Z -1.3333, A 0.000, B 0.000, C 0.000 }
gfCNCPoint1[17951] = {X 7.6640, Y 35.3085, Z -1.3333, A 0.000, B 0.000, C 0.000 }
gfCNCPoint1[17952] = {X 7.6543, Y 35.3707, Z -1.3333, A 0.000, B 0.000, C 0.000 }
gfCNCPoint1[17953] = {X 7.6509, Y 35.4334, Z -1.3333, A 0.000, B 0.000, C 0.000 }
gfCNCPoint1[17954] = {X 7.7517, Y 36.0270, Z -1.3333, A 0.000, B 0.000, C 0.000 }
gfCNCPoint1[17955] = {X 8.0468, Y 36.5519, Z -1.3333, A 0.000, B 0.000, C 0.000 }
gfCNCPoint1[17956] = {X 8.5015, Y 36.9465, Z -1.3333, A 0.000, B 0.000, C 0.000 }
gfCNCPoint1[17957] = {X 9.2748, Y 37.3380, Z -1.3333, A 0.000, B 0.000, C 0.000 }
gfCNCPoint1[17958] = {X 10.0975, Y 37.6108, Z -1.3333, A 0.000, B 0.000, C 0.000 }
gfCNCPoint1[17959] = {X 11.3746, Y 37.8475, Z -1.3333, A 0.000, B 0.000, C 0.000 }
gfCNCPoint1[17960] = {X 12.6714, Y 37.9226, Z -1.3333, A 0.000, B 0.000, C 0.000 }
gfCNCPoint1[17961] = {X 13.9673, Y 37.8346, Z -1.3333, A 0.000, B 0.000, C 0.000 }
gfCNCPoint1[17962] = {X 15.2420, Y 37.5852, Z -1.3333, A 0.000, B 0.000, C 0.000 }
gfCNCPoint1[17963] = {X 16.4755, Y 37.1782, Z -1.3333, A 0.000, B 0.000, C 0.000 }
gfCNCPoint1[17964] = {X 17.7922, Y 36.5649, Z -1.3333, A 0.000, B 0.000, C 0.000 }
gfCNCPoint1[17965] = {X 19.0345, Y 35.8124, Z -1.3333, A 0.000, B 0.000, C 0.000 }
gfCNCPoint1[17966] = {X 19.1548, Y 34.9704, Z -1.3333, A 0.000, B 0.000, C 0.000 }
gfCNCPoint1[17967] = {X 19.4349, Y 34.1672, Z -1.3333, A 0.000, B 0.000, C 0.000 }
gfCNCPoint1[17968] = {X 17.7799, Y 34.4451, Z -1.3333, A 0.000, B 0.000, C 0.000 }
gfCNCPoint1[17969] = {X 16.1107, Y 34.6182, Z -1.3333, A 0.000, B 0.000, C 0.000 }
gfCNCPoint1[17970] = {X 15.3860, Y 34.6709, Z -1.3333, A 0.000, B 0.000, C 0.000 }
gfCNCPoint1[17971] = {X 14.6611, Y 34.7215, Z -1.3333, A 0.000, B 0.000, C 0.000 }
gfCNCPoint1[17972] = {X 18.6550, Y 34.7177, Z -1.3333, A 0.000, B 0.000, C 0.000 }
gfCNCPoint1[17973] = {X 14.6557, Y 34.6417, Z -1.3333, A 0.000, B 0.000, C 0.000 }
gfCNCPoint1[17974] = {X 12.2591, Y 34.7942, Z -1.3333, A 0.000, B 0.000, C 0.000 }
gfCNCPoint1[17975] = {X 9.8611, Y 34.9238, Z -1.3333, A 0.000, B 0.000, C 0.000 }
gfCNCPoint1[17976] = {X 8.7202, Y 35.0182, Z -1.3333, A 0.000, B 0.000, C 0.000 }
gfCNCPoint1[17977] = {X 7.5978, Y 35.2430, Z -1.3333, A 0.000, B 0.000, C 0.000 }
gfCNCPoint1[17978] = {X 7.5778, Y 35.3372, Z -1.3333, A 0.000, B 0.000, C 0.000 }
gfCNCPoint1[17979] = {X 7.5709, Y 35.4331, Z -1.3333, A 0.000, B 0.000, C 0.000 }
gfCNCPoint1[17980] = {X 7.6763, Y 36.0537, Z -1.3333, A 0.000, B 0.000, C 0.000 }
gfCNCPoint1[17981] = {X 7.9848, Y 36.6024, Z -1.3333, A 0.000, B 0.000, C 0.000 }
gfCNCPoint1[17982] = {X 8.4602, Y 37.0150, Z -1.3333, A 0.000, B 0.000, C 0.000 }
gfCNCPoint1[17983] = {X 9.2441, Y 37.4118, Z -1.3333, A 0.000, B 0.000, C 0.000 }
gfCNCPoint1[17984] = {X 10.0780, Y 37.6884, Z -1.3333, A 0.000, B 0.000, C 0.000 }
gfCNCPoint1[17985] = {X 11.3650, Y 37.9270, Z -1.3333, A 0.000, B 0.000, C 0.000 }
gfCNCPoint1[17986] = {X 12.6718, Y 38.0026, Z -1.3333, A 0.000, B 0.000, C 0.000 }
gfCNCPoint1[17987] = {X 13.9777, Y 37.9140, Z -1.3333, A 0.000, B 0.000, C 0.000 }
gfCNCPoint1[17988] = {X 15.2623, Y 37.6626, Z -1.3333, A 0.000, B 0.000, C 0.000 }
gfCNCPoint1[17989] = {X 16.5053, Y 37.2524, Z -1.3333, A 0.000, B 0.000, C 0.000 }
gfCNCPoint1[17990] = {X 17.8476, Y 36.6260, Z -1.3333, A 0.000, B 0.000, C 0.000 }
gfCNCPoint1[17991] = {X 19.1128, Y 35.8558, Z -1.3333, A 0.000, B 0.000, C 0.000 }
gfCNCPoint1[17992] = {X 19.2472, Y 34.9309, Z -1.3333, A 0.000, B 0.000, C 0.000 }
gfCNCPoint1[17993] = {X 19.5774, Y 34.0565, Z -1.3333, A 0.000, B 0.000, C 0.000 }
gfCNCPoint1[17994] = {X 17.8491, Y 34.3549, Z -1.3333, A 0.000, B 0.000, C 0.000 }
gfCNCPoint1[17995] = {X 16.1049, Y 34.5384, Z -1.3333, A 0.000, B 0.000, C 0.000 }
gfCNCPoint1[17996] = {X 15.3804, Y 34.5911, Z -1.3333, A 0.000, B 0.000, C 0.000 }
gfCNCPoint1[17997] = {X 14.6557, Y 34.6417, Z -1.3333, A 0.000, B 0.000, C 0.000 }
gfCNCPoint1[17998] = {X 10.7040, Y 35.2614, Z -1.3333, A 0.000, B 0.000, C 0.000 }
gfCNCPoint1[17999] = {X 18.6495, Y 34.6379, Z -1.3333, A 0.000, B 0.000, C 0.000 }
gfCNCPoint1[18000] = {X 14.6502, Y 34.5619, Z -1.3333, A 0.000, B 0.000, C 0.000 }
gfCNCPoint1[18001] = {X 12.2549, Y 34.7143, Z -1.3333, A 0.000, B 0.000, C 0.000 }
gfCNCPoint1[18002] = {X 9.8582, Y 34.8438, Z -1.3333, A 0.000, B 0.000, C 0.000 }
gfCNCPoint1[18003] = {X 8.6867, Y 34.9421, Z -1.3333, A 0.000, B 0.000, C 0.000 }
gfCNCPoint1[18004] = {X 7.5348, Y 35.1769, Z -1.3333, A 0.000, B 0.000, C 0.000 }
gfCNCPoint1[18005] = {X 7.5022, Y 35.3030, Z -1.3333, A 0.000, B 0.000, C 0.000 }
gfCNCPoint1[18006] = {X 7.4909, Y 35.4328, Z -1.3333, A 0.000, B 0.000, C 0.000 }
gfCNCPoint1[18007] = {X 7.6009, Y 36.0804, Z -1.3333, A 0.000, B 0.000, C 0.000 }
gfCNCPoint1[18008] = {X 7.9228, Y 36.6530, Z -1.3333, A 0.000, B 0.000, C 0.000 }
gfCNCPoint1[18009] = {X 8.4189, Y 37.0835, Z -1.3333, A 0.000, B 0.000, C 0.000 }
gfCNCPoint1[18010] = {X 9.2133, Y 37.4857, Z -1.3333, A 0.000, B 0.000, C 0.000 }
gfCNCPoint1[18011] = {X 10.0585, Y 37.7660, Z -1.3333, A 0.000, B 0.000, C 0.000 }
gfCNCPoint1[18012] = {X 11.3554, Y 38.0064, Z -1.3333, A 0.000, B 0.000, C 0.000 }
gfCNCPoint1[18013] = {X 12.6722, Y 38.0826, Z -1.3333, A 0.000, B 0.000, C 0.000 }
gfCNCPoint1[18014] = {X 13.9881, Y 37.9933, Z -1.3333, A 0.000, B 0.000, C 0.000 }
gfCNCPoint1[18015] = {X 15.2826, Y 37.7400, Z -1.3333, A 0.000, B 0.000, C 0.000 }
gfCNCPoint1[18016] = {X 16.5351, Y 37.3267, Z -1.3333, A 0.000, B 0.000, C 0.000 }
gfCNCPoint1[18017] = {X 17.9032, Y 36.6870, Z -1.3333, A 0.000, B 0.000, C 0.000 }
gfCNCPoint1[18018] = {X 19.1915, Y 35.8987, Z -1.3333, A 0.000, B 0.000, C 0.000 }
gfCNCPoint1[18019] = {X 19.2643, Y 35.2207, Z -1.3333, A 0.000, B 0.000, C 0.000 }
gfCNCPoint1[18020] = {X 19.4448, Y 34.5631, Z -1.3333, A 0.000, B 0.000, C 0.000 }
gfCNCPoint1[18021] = {X 19.7285, Y 33.9430, Z -1.3333, A 0.000, B 0.000, C 0.000 }
gfCNCPoint1[18022] = {X 17.9227, Y 34.2638, Z -1.3333, A 0.000, B 0.000, C 0.000 }
gfCNCPoint1[18023] = {X 16.0991, Y 34.4586, Z -1.3333, A 0.000, B 0.000, C 0.000 }
gfCNCPoint1[18024] = {X 15.3747, Y 34.5113, Z -1.3333, A 0.000, B 0.000, C 0.000 }
gfCNCPoint1[18025] = {X 14.6502, Y 34.5619, Z -1.3333, A 0.000, B 0.000, C 0.000 }
gfCNCPoint1[18026] = {X 10.6985, Y 35.1816, Z -1.3333, A 0.000, B 0.000, C 0.000 }
gfCNCPoint1[18027] = {X 18.6440, Y 34.5581, Z -1.3333, A 0.000, B 0.000, C 0.000 }
gfCNCPoint1[18028] = {X 14.6448, Y 34.4821, Z -1.3333, A 0.000, B 0.000, C 0.000 }
gfCNCPoint1[18029] = {X 12.2506, Y 34.6344, Z -1.3333, A 0.000, B 0.000, C 0.000 }
gfCNCPoint1[18030] = {X 9.8552, Y 34.7639, Z -1.3333, A 0.000, B 0.000, C 0.000 }
gfCNCPoint1[18031] = {X 8.6545, Y 34.8660, Z -1.3333, A 0.000, B 0.000, C 0.000 }
gfCNCPoint1[18032] = {X 7.4745, Y 35.1102, Z -1.3333, A 0.000, B 0.000, C 0.000 }
gfCNCPoint1[18033] = {X 7.4273, Y 35.2683, Z -1.3333, A 0.000, B 0.000, C 0.000 }
gfCNCPoint1[18034] = {X 7.4109, Y 35.4326, Z -1.3333, A 0.000, B 0.000, C 0.000 }
gfCNCPoint1[18035] = {X 7.5255, Y 36.1071, Z -1.3333, A 0.000, B 0.000, C 0.000 }
